KUKA KRL program: MyProgram_279().src

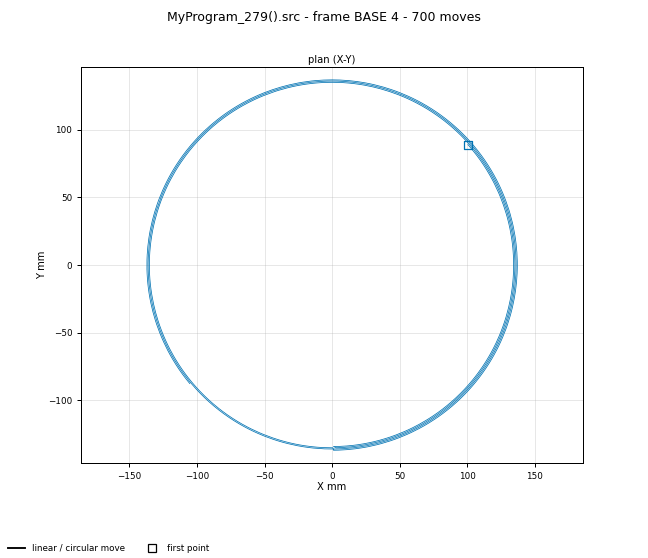
[picture p0: tool path of MyProgram_279().src in frame BASE 4, 700 of 700 moves have a stored position in this frame; points joined in program order, loops and branches not executed]
&ACCESS RVP
&REL 1
&PARAM TEMPLATE = C:\KRC\Roboter\Template\vorgabe
&PARAM EDITMASK = *
DEF MyProgram_279()
; ---- Setting reference (Base) ----
$BASE = BASE_DATA[4]

; --------------------------
; ---- Setting tool (TCP) ----
$TOOL = TOOL_DATA[3]
; --------------------------

$VEL.CP = VEL_APROX_PRINT
Startdeposition()
$VEL.CP = VEL_PRINT
LIN {X 100.485,Y 89.1473,Z 173,A 42.0172,B 8.5894,C 0.1342,E1 8.7113,E2 409.55} C_DIS
LIN {X 102.9839,Y 86.2482,Z 173,A 40.2493,B 8.5893,C 0.1406,E1 8.7146,E2 411.3348} C_DIS
LIN {X 107.2728,Y 80.8516,Z 173,A 37.5079,B 8.5893,C 0.1431,E1 8.7192,E2 414.0536} C_DIS
LIN {X 109.4869,Y 77.827,Z 173,A 35.923,B 8.5892,C 0.1466,E1 8.7218,E2 415.6375} C_DIS
LIN {X 111.988,Y 74.1839,Z 173,A 34.0395,B 8.5891,C 0.151,E1 8.7248,E2 417.5218} C_DIS
LIN {X 114.278,Y 70.6054,Z 173,A 32.2397,B 8.5891,C 0.1552,E1 8.7274,E2 419.3211} C_DIS
LIN {X 116.5443,Y 66.7977,Z 173,A 30.3906,B 8.5889,C 0.159,E1 8.73,E2 421.1663} C_DIS
LIN {X 118.6905,Y 62.9024,Z 173,A 28.6674,B 8.5889,C 0.1602,E1 8.7323,E2 422.8695} C_DIS
LIN {X 120.2957,Y 59.7744,Z 173,A 27.1057,B 8.5889,C 0.1653,E1 8.7343,E2 424.4396} C_DIS
LIN {X 121.8682,Y 56.4983,Z 173,A 25.7054,B 8.5889,C 0.1662,E1 8.7359,E2 425.8228} C_DIS
LIN {X 123.1677,Y 53.6072,Z 173,A 24.298,B 8.5887,C 0.171,E1 8.7375,E2 427.2377} C_DIS
LIN {X 124.4105,Y 50.6572,Z 173,A 23.0997,B 8.5887,C 0.171,E1 8.7388,E2 428.4167} C_DIS
LIN {X 126.8287,Y 44.2546,Z 173,A 20.1497,B 8.5885,C 0.1796,E1 8.7417,E2 431.3725} C_DIS
LIN {X 127.8957,Y 41.0691,Z 173,A 18.3823,B 8.5883,C 0.1906,E1 8.7432,E2 433.1816} C_DIS
LIN {X 128.857,Y 37.9453,Z 173,A 17.2852,B 8.5883,C 0.1882,E1 8.7441,E2 434.2437} C_DIS
LIN {X 129.7659,Y 34.7098,Z 173,A 15.8546,B 8.5883,C 0.1921,E1 8.7451,E2 435.675} C_DIS
LIN {X 130.7274,Y 30.8976,Z 173,A 14.1088,B 8.5881,C 0.1983,E1 8.7463,E2 437.4306} C_DIS
LIN {X 131.5915,Y 26.9758,Z 173,A 12.5684,B 8.5881,C 0.1994,E1 8.7472,E2 438.9513} C_DIS
LIN {X 132.2101,Y 23.7589,Z 173,A 11.1939,B 8.5881,C 0.2029,E1 8.7479,E2 440.3242} C_DIS
LIN {X 132.7584,Y 20.4746,Z 173,A 9.8483,B 8.588,C 0.2054,E1 8.7485,E2 441.6618} C_DIS
LIN {X 133.24,Y 17.0665,Z 173,A 8.3029,B 8.5878,C 0.2112,E1 8.7491,E2 443.2179} C_DIS
LIN {X 133.6974,Y 13.002,Z 173,A 6.6491,B 8.5878,C 0.2143,E1 8.7496,E2 444.8621} C_DIS
LIN {X 133.9613,Y 9.9205,Z 173,A 5.3303,B 8.5877,C 0.2181,E1 8.7498,E2 446.182} C_DIS
LIN {X 134.1788,Y 6.3448,Z 173,A 3.8957,B 8.5876,C 0.2205,E1 8.7501,E2 447.6065} C_DIS
LIN {X 134.3024,Y 2.6623,Z 173,A 2.2339,B 8.5874,C 0.227,E1 8.7501,E2 449.2808} C_DIS
LIN {X 134.324,Y -1.2062,Z 173,A 0.5555,B 8.5873,C 0.2324,E1 8.7501,E2 450.9642} C_DIS
LIN {X 134.2251,Y -5.2587,Z 173,A -1.0909,B 8.5872,C 0.2356,E1 8.7501,E2 452.602} C_DIS
LIN {X 133.985,Y -9.596,Z 173,A -2.8654,B 8.5871,C 0.2393,E1 8.7497,E2 454.3687} C_DIS
LIN {X 133.6414,Y -13.585,Z 173,A -4.6499,B 8.5869,C 0.2459,E1 8.7493,E2 456.1642} C_DIS
LIN {X 133.1911,Y -17.4395,Z 173,A -6.1529,B 8.5869,C 0.2474,E1 8.7488,E2 457.6502} C_DIS
LIN {X 132.6837,Y -20.9568,Z 173,A -7.6551,B 8.5867,C 0.2515,E1 8.7481,E2 459.1521} C_DIS
LIN {X 131.966,Y -25.0793,Z 173,A -9.4147,B 8.5867,C 0.2561,E1 8.7473,E2 460.9104} C_DIS
LIN {X 131.3008,Y -28.3563,Z 173,A -10.761,B 8.5865,C 0.2584,E1 8.7465,E2 462.2482} C_DIS
LIN {X 130.5715,Y -31.5445,Z 173,A -12.2103,B 8.5864,C 0.2636,E1 8.7456,E2 463.7057} C_DIS
LIN {X 128.6891,Y -38.5187,Z 173,A -15.3512,B 8.5861,C 0.2735,E1 8.7432,E2 466.8571} C_DIS
LIN {X 127.5485,Y -42.1357,Z 173,A -16.8717,B 8.5861,C 0.276,E1 8.7419,E2 468.3673} C_DIS
LIN {X 126.1394,Y -46.1868,Z 173,A -18.7317,B 8.5858,C 0.2817,E1 8.7402,E2 470.2329} C_DIS
LIN {X 124.7098,Y -49.9148,Z 173,A -20.2936,B 8.5858,C 0.2833,E1 8.7386,E2 471.7791} C_DIS
LIN {X 123.4262,Y -53.0093,Z 173,A -21.6078,B 8.5858,C 0.2847,E1 8.7372,E2 473.0806} C_DIS
LIN {X 121.271,Y -57.7684,Z 173,A -24.375,B 8.5851,C 0.3021,E1 8.7338,E2 475.9163} C_DIS
LIN {X 119.2793,Y -61.7811,Z 173,A -25.7267,B 8.5854,C 0.2953,E1 8.7322,E2 477.2014} C_DIS
LIN {X 117.6517,Y -64.8271,Z 173,A -27.5786,B 8.585,C 0.3071,E1 8.7297,E2 479.1015} C_DIS
LIN {X 115.8509,Y -67.9927,Z 173,A -28.7916,B 8.585,C 0.3039,E1 8.728,E2 480.2742} C_DIS
LIN {X 113.7196,Y -71.5006,Z 173,A -30.5786,B 8.5849,C 0.3091,E1 8.7254,E2 482.0674} C_DIS
LIN {X 111.2545,Y -75.2785,Z 173,A -33.0154,B 8.5843,C 0.3245,E1 8.7215,E2 484.5691} C_DIS
LIN {X 108.269,Y -79.5126,Z 173,A -34.9644,B 8.5843,C 0.3245,E1 8.7183,E2 486.4884} C_DIS
LIN {X 105.8625,Y -82.6903,Z 173,A -36.3361,B 8.5844,C 0.3216,E1 8.716,E2 487.8214} C_DIS
LIN {X 103.7415,Y -85.3365,Z 173,A -37.6368,B 8.5844,C 0.3219,E1 8.7138,E2 489.1056} C_DIS
LIN {X 100.7739,Y -88.8205,Z 173,A -39.6561,B 8.5842,C 0.3277,E1 8.7101,E2 491.1352} C_DIS
LIN {X 97.9294,Y -91.9476,Z 173,A -41.4693,B 8.584,C 0.3319,E1 8.7066,E2 492.9514} C_DIS
LIN {X 94.9858,Y -94.9858,Z 173,A -43.1042,B 8.584,C 0.3322,E1 8.7035,E2 494.5671} C_DIS
LIN {X 91.8309,Y -98.0391,Z 173,A -45.1099,B 8.5838,C 0.3389,E1 8.6994,E2 496.5911} C_DIS
LIN {X 88.4514,Y -101.098,Z 173,A -47.0097,B 8.5837,C 0.3418,E1 8.6954,E2 498.4872} C_DIS
LIN {X 84.9527,Y -104.0551,Z 173,A -48.6273,B 8.5837,C 0.3387,E1 8.6921,E2 500.065} C_DIS
LIN {X 81.7579,Y -106.5834,Z 173,A -50.7305,B 8.5833,C 0.3495,E1 8.6873,E2 502.2152} C_DIS
LIN {X 78.4256,Y -109.0596,Z 173,A -52.5118,B 8.5833,C 0.3529,E1 8.6833,E2 503.9994} C_DIS
LIN {X 74.2386,Y -111.9519,Z 173,A -54.5479,B 8.5832,C 0.3539,E1 8.6786,E2 506.0209} C_DIS
LIN {X 70.5082,Y -114.3377,Z 173,A -56.5951,B 8.5829,C 0.3601,E1 8.6737,E2 508.0893} C_DIS
LIN {X 64.3845,Y -117.8942,Z 173,A -59.5316,B 8.5828,C 0.3631,E1 8.6666,E2 511.018} C_DIS
LIN {X 59.9186,Y -120.2246,Z 173,A -61.4357,B 8.5828,C 0.3613,E1 8.6619,E2 512.8936} C_DIS
LIN {X 56.6377,Y -121.8037,Z 173,A -62.9476,B 8.5828,C 0.3625,E1 8.6581,E2 514.4015} C_DIS
LIN {X 53.5188,Y -123.2059,Z 173,A -64.428,B 8.5828,C 0.3648,E1 8.6543,E2 515.8858} C_DIS
LIN {X 50.3544,Y -124.5326,Z 173,A -65.8538,B 8.5827,C 0.3658,E1 8.6507,E2 517.3081} C_DIS
LIN {X 47.4368,Y -125.6733,Z 173,A -67.113,B 8.5827,C 0.3658,E1 8.6474,E2 518.5588} C_DIS
LIN {X 43.2176,Y -127.1882,Z 173,A -69.2595,B 8.5824,C 0.3725,E1 8.6417,E2 520.736} C_DIS
LIN {X 39.3019,Y -128.4496,Z 173,A -70.9006,B 8.5824,C 0.372,E1 8.6373,E2 522.3641} C_DIS
LIN {X 35.3098,Y -129.6059,Z 173,A -72.676,B 8.5824,C 0.3737,E1 8.6326,E2 524.1412} C_DIS
LIN {X 31.6272,Y -130.5515,Z 173,A -74.2847,B 8.5823,C 0.3748,E1 8.6282,E2 525.7494} C_DIS
LIN {X 27.725,Y -131.437,Z 173,A -75.9912,B 8.5823,C 0.376,E1 8.6235,E2 527.4569} C_DIS
LIN {X 23.8324,Y -132.1969,Z 173,A -77.6907,B 8.5822,C 0.3773,E1 8.6189,E2 529.1585} C_DIS
LIN {X 19.6935,Y -132.8783,Z 173,A -79.4646,B 8.5822,C 0.378,E1 8.614,E2 530.9316} C_DIS
LIN {X 15.995,Y -133.3723,Z 173,A -81.0275,B 8.5822,C 0.3782,E1 8.6097,E2 532.4918} C_DIS
LIN {X 10.8636,Y -133.8887,Z 173,A -83.2675,B 8.5821,C 0.3799,E1 8.6034,E2 534.7381} C_DIS
LIN {X 4.7872,Y -134.2435,Z 173,A -85.8421,B 8.5821,C 0.3802,E1 8.5962,E2 537.3113} C_DIS
LIN {X 0.9731,Y -134.3248,Z 173,A -87.1721,B 8.5823,C 0.3749,E1 8.5926,E2 538.6052} C_DIS
Enddeposition()
LIN {X 0.9731,Y -134.3248,Z 173,A -87.1721,B 8.5823,C 0.3749,E1 8.5926,E2 538.6052} C_DIS
Startdeposition()
$VEL.CP = VEL_PRINT
LIN {X 3.1797,Y -135.2005,Z 173,A -85.0351,B 8.4211,C 0.3601,E1 8.4372,E2 536.3964} C_DIS
LIN {X 8.6007,Y -134.9631,Z 173,A -83.5881,B 8.4204,C 0.3756,E1 8.4409,E2 535.0567} C_DIS
LIN {X 14.6467,Y -134.4411,Z 173,A -80.9054,B 8.4206,C 0.3725,E1 8.4484,E2 532.3585} C_DIS
LIN {X 18.2658,Y -133.9991,Z 173,A -79.1927,B 8.4208,C 0.3685,E1 8.4532,E2 530.6237} C_DIS
LIN {X 22.5658,Y -133.3408,Z 173,A -77.3912,B 8.4208,C 0.3682,E1 8.4581,E2 528.8263} C_DIS
LIN {X 26.9688,Y -132.52,Z 173,A -75.6345,B 8.4208,C 0.3697,E1 8.4629,E2 527.0862} C_DIS
LIN {X 30.1469,Y -131.8334,Z 173,A -74.2295,B 8.4208,C 0.3681,E1 8.4667,E2 525.6768} C_DIS
LIN {X 33.3306,Y -131.0646,Z 173,A -72.832,B 8.4208,C 0.3668,E1 8.4705,E2 524.2772} C_DIS
LIN {X 37.4094,Y -129.9606,Z 173,A -71.0032,B 8.4209,C 0.3644,E1 8.4755,E2 522.4423} C_DIS
LIN {X 41.0365,Y -128.8598,Z 173,A -69.4333,B 8.4209,C 0.3636,E1 8.4796,E2 520.8757} C_DIS
LIN {X 45.0729,Y -127.5065,Z 173,A -67.7068,B 8.4209,C 0.3632,E1 8.4842,E2 519.1578} C_DIS
LIN {X 48.3644,Y -126.294,Z 173,A -66.2819,B 8.421,C 0.3627,E1 8.4879,E2 517.7394} C_DIS
LIN {X 50.929,Y -125.2805,Z 173,A -65.0721,B 8.421,C 0.3605,E1 8.491,E2 516.5235} C_DIS
LIN {X 53.8536,Y -124.0509,Z 173,A -63.7005,B 8.4212,C 0.3583,E1 8.4946,E2 515.1473} C_DIS
LIN {X 57.7786,Y -122.2733,Z 173,A -62.0162,B 8.4212,C 0.3587,E1 8.4988,E2 513.4794} C_DIS
LIN {X 61.6591,Y -120.3622,Z 173,A -60.1136,B 8.4213,C 0.3547,E1 8.5036,E2 511.5664} C_DIS
LIN {X 66.6135,Y -117.6943,Z 173,A -57.6159,B 8.4216,C 0.3489,E1 8.5097,E2 509.0523} C_DIS
LIN {X 70.7017,Y -115.2849,Z 173,A -55.6539,B 8.4216,C 0.3467,E1 8.5144,E2 507.0947} C_DIS
LIN {X 74.6014,Y -112.8009,Z 173,A -53.7083,B 8.4218,C 0.3437,E1 8.519,E2 505.1492} C_DIS
LIN {X 78.6189,Y -110.0383,Z 173,A -51.7429,B 8.4218,C 0.3421,E1 8.5235,E2 503.1945} C_DIS
LIN {X 81.7657,Y -107.7212,Z 173,A -49.6484,B 8.4223,C 0.3301,E1 8.5283,E2 501.0428} C_DIS
LIN {X 85.0887,Y -105.1157,Z 173,A -48.2843,B 8.4221,C 0.3354,E1 8.5311,E2 499.731} C_DIS
LIN {X 88.4159,Y -102.3328,Z 173,A -46.4652,B 8.4223,C 0.3322,E1 8.535,E2 497.9126} C_DIS
LIN {X 91.7629,Y -99.3429,Z 173,A -44.5493,B 8.4224,C 0.3281,E1 8.5389,E2 495.993} C_DIS
LIN {X 95.6283,Y -95.6283,Z 173,A -42.418,B 8.4224,C 0.3262,E1 8.5432,E2 493.8773} C_DIS
LIN {X 98.3275,Y -92.8496,Z 173,A -40.7262,B 8.4227,C 0.3216,E1 8.5465,E2 492.1774} C_DIS
LIN {X 101.0457,Y -89.8848,Z 173,A -39.0307,B 8.4227,C 0.318,E1 8.5496,E2 490.4813} C_DIS
LIN {X 104.5568,Y -85.7745,Z 173,A -36.7353,B 8.423,C 0.3127,E1 8.5538,E2 488.183} C_DIS
LIN {X 108.0978,Y -81.2666,Z 173,A -34.3605,B 8.4232,C 0.3081,E1 8.5578,E2 485.8126} C_DIS
LIN {X 111.5883,Y -76.403,Z 173,A -32.212,B 8.4231,C 0.3101,E1 8.5612,E2 483.7105} C_DIS
LIN {X 114.2276,Y -72.398,Z 173,A -29.8489,B 8.4235,C 0.2981,E1 8.5649,E2 481.3037} C_DIS
LIN {X 116.5329,Y -68.6255,Z 173,A -27.7284,B 8.4239,C 0.2881,E1 8.5679,E2 479.1499} C_DIS
LIN {X 118.4042,Y -65.344,Z 173,A -26.6704,B 8.4236,C 0.2955,E1 8.5693,E2 478.1588} C_DIS
LIN {X 119.9038,Y -62.5461,Z 173,A -25.1858,B 8.4238,C 0.289,E1 8.5713,E2 476.6552} C_DIS
LIN {X 121.4823,Y -59.4226,Z 173,A -22.9203,B 8.4245,C 0.2684,E1 8.5742,E2 474.2889} C_DIS
LIN {X 124.0675,Y -53.8154,Z 173,A -21.4335,B 8.424,C 0.2855,E1 8.5757,E2 472.9424} C_DIS
LIN {X 125.5947,Y -50.1496,Z 173,A -19.5623,B 8.4242,C 0.277,E1 8.5777,E2 471.0459} C_DIS
LIN {X 126.6911,Y -47.3097,Z 173,A -18.1837,B 8.4244,C 0.2715,E1 8.5791,E2 469.6547} C_DIS
LIN {X 127.9892,Y -43.681,Z 173,A -16.684,B 8.4244,C 0.2699,E1 8.5804,E2 468.1702} C_DIS
LIN {X 128.9127,Y -40.871,Z 173,A -15.3598,B 8.4246,C 0.2648,E1 8.5816,E2 466.8357} C_DIS
LIN {X 130.0092,Y -37.2433,Z 173,A -13.0796,B 8.4252,C 0.2458,E1 8.5834,E2 464.4687} C_DIS
LIN {X 131.459,Y -31.7395,Z 173,A -11.7613,B 8.4247,C 0.2625,E1 8.5842,E2 463.2858} C_DIS
LIN {X 132.4574,Y -27.2767,Z 173,A -9.5172,B 8.4251,C 0.2504,E1 8.5856,E2 461.0015} C_DIS
LIN {X 133.2044,Y -23.3604,Z 173,A -7.7659,B 8.4252,C 0.2443,E1 8.5864,E2 459.2407} C_DIS
LIN {X 133.8801,Y -19.1054,Z 173,A -6.0865,B 8.4253,C 0.2422,E1 8.5871,E2 457.5779} C_DIS
LIN {X 134.3319,Y -15.6208,Z 173,A -4.6379,B 8.4253,C 0.2387,E1 8.5876,E2 456.1329} C_DIS
LIN {X 134.7345,Y -11.6447,Z 173,A -2.9675,B 8.4255,C 0.2343,E1 8.5881,E2 454.4637} C_DIS
LIN {X 134.9923,Y -8.1275,Z 173,A -1.3919,B 8.4257,C 0.2282,E1 8.5884,E2 452.8765} C_DIS
LIN {X 135.1862,Y -3.6953,Z 173,A 0.338,B 8.4257,C 0.226,E1 8.5885,E2 451.1636} C_DIS
LIN {X 135.2394,Y 0.1311,Z 173,A 2.0503,B 8.4259,C 0.2194,E1 8.5885,E2 449.4386} C_DIS
LIN {X 135.1662,Y 4.4152,Z 173,A 3.7592,B 8.4259,C 0.2164,E1 8.5885,E2 447.7414} C_DIS
LIN {X 134.9832,Y 8.2747,Z 173,A 5.3221,B 8.4261,C 0.2132,E1 8.5882,E2 446.1862} C_DIS
LIN {X 134.7234,Y 11.7761,Z 173,A 6.8793,B 8.4262,C 0.2075,E1 8.5878,E2 444.619} C_DIS
LIN {X 134.2911,Y 15.9626,Z 173,A 8.5658,B 8.4262,C 0.2044,E1 8.5873,E2 442.943} C_DIS
LIN {X 133.7903,Y 19.734,Z 173,A 10.2222,B 8.4264,C 0.1989,E1 8.5867,E2 441.2797} C_DIS
LIN {X 133.1155,Y 23.8569,Z 173,A 11.8788,B 8.4264,C 0.1962,E1 8.5859,E2 439.6358} C_DIS
LIN {X 132.477,Y 27.1805,Z 173,A 13.2505,B 8.4266,C 0.1935,E1 8.5852,E2 438.2706} C_DIS
LIN {X 131.6646,Y 30.8858,Z 173,A 14.9649,B 8.4267,C 0.1867,E1 8.5841,E2 436.5417} C_DIS
LIN {X 130.706,Y 34.7103,Z 173,A 16.4987,B 8.4267,C 0.1849,E1 8.583,E2 435.0236} C_DIS
LIN {X 129.7458,Y 38.1432,Z 173,A 18.322,B 8.427,C 0.1741,E1 8.5816,E2 433.1602} C_DIS
LIN {X 128.6869,Y 41.578,Z 173,A 19.5895,B 8.427,C 0.1754,E1 8.5805,E2 431.9235} C_DIS
LIN {X 126.9178,Y 46.6997,Z 173,A 22.0901,B 8.4272,C 0.1648,E1 8.5781,E2 429.3957} C_DIS
LIN {X 125.6176,Y 50.0929,Z 173,A 23.1235,B 8.427,C 0.1714,E1 8.5772,E2 428.4242} C_DIS
LIN {X 123.9922,Y 53.9895,Z 173,A 24.9665,B 8.4271,C 0.1655,E1 8.5751,E2 426.5732} C_DIS
LIN {X 122.6804,Y 56.9065,Z 173,A 26.3336,B 8.4272,C 0.1617,E1 8.5735,E2 425.2039} C_DIS
LIN {X 121.1858,Y 60.0236,Z 173,A 27.7918,B 8.4272,C 0.158,E1 8.5718,E2 423.7455} C_DIS
LIN {X 119.6303,Y 63.0669,Z 173,A 29.1984,B 8.4273,C 0.1552,E1 8.57,E2 422.3432} C_DIS
LIN {X 117.6594,Y 66.6765,Z 173,A 31.0566,B 8.4275,C 0.1484,E1 8.5674,E2 420.4698} C_DIS
LIN {X 115.435,Y 70.457,Z 173,A 32.8581,B 8.4275,C 0.1451,E1 8.5648,E2 418.6744} C_DIS
LIN {X 113.1585,Y 74.0582,Z 173,A 34.6628,B 8.4275,C 0.1407,E1 8.5621,E2 416.8687} C_DIS
LIN {X 110.5824,Y 77.8516,Z 173,A 36.3712,B 8.4275,C 0.141,E1 8.5594,E2 415.1882} C_DIS
LIN {X 108.5001,Y 80.7283,Z 173,A 38.0366,B 8.4277,C 0.1342,E1 8.5566,E2 413.5023} C_DIS
LIN {X 104.2889,Y 86.1,Z 173,A 40.7446,B 8.4277,C 0.1315,E1 8.552,E2 410.8158} C_DIS
LIN {X 101.8703,Y 88.9481,Z 173,A 42.4537,B 8.4278,C 0.1255,E1 8.5488,E2 409.0907} C_DIS
LIN {X 98.7737,Y 92.3752,Z 173,A 44.3706,B 8.4278,C 0.1221,E1 8.5452,E2 407.178} C_DIS
LIN {X 95.502,Y 95.7537,Z 173,A 46.2585,B 8.4279,C 0.1202,E1 8.5415,E2 405.3023} C_DIS
LIN {X 92.5535,Y 98.6068,Z 173,A 48.0619,B 8.4279,C 0.1154,E1 8.5379,E2 403.4904} C_DIS
LIN {X 89.182,Y 101.6663,Z 173,A 49.991,B 8.428,C 0.1118,E1 8.5339,E2 401.5607} C_DIS
LIN {X 85.7804,Y 104.552,Z 173,A 51.8548,B 8.428,C 0.1088,E1 8.5299,E2 399.6997} C_DIS
LIN {X 82.3114,Y 107.3043,Z 173,A 53.6976,B 8.428,C 0.1062,E1 8.5258,E2 397.8607} C_DIS
LIN {X 78.8304,Y 109.887,Z 173,A 55.5035,B 8.4281,C 0.1037,E1 8.5217,E2 396.0582} C_DIS
LIN {X 74.0069,Y 113.1923,Z 173,A 57.9951,B 8.4281,C 0.0995,E1 8.516,E2 393.5646} C_DIS
LIN {X 70.2078,Y 115.5867,Z 173,A 59.8837,B 8.4282,C 0.0969,E1 8.5115,E2 391.6775} C_DIS
LIN {X 66.4641,Y 117.7791,Z 173,A 61.6957,B 8.4282,C 0.0948,E1 8.5071,E2 389.8686} C_DIS
LIN {X 62.5875,Y 119.882,Z 173,A 63.4373,B 8.4282,C 0.0948,E1 8.5029,E2 388.1424} C_DIS
LIN {X 59.215,Y 121.5847,Z 173,A 65.0144,B 8.4282,C 0.0931,E1 8.4989,E2 386.5682} C_DIS
LIN {X 55.8747,Y 123.1557,Z 173,A 66.6829,B 8.4282,C 0.0893,E1 8.4946,E2 384.887} C_DIS
LIN {X 52.258,Y 124.7314,Z 173,A 68.2626,B 8.4282,C 0.0891,E1 8.4906,E2 383.3186} C_DIS
LIN {X 49.0309,Y 126.0349,Z 173,A 69.5241,B 8.4282,C 0.0916,E1 8.4874,E2 382.0831} C_DIS
LIN {X 45.1831,Y 127.467,Z 173,A 71.4243,B 8.4283,C 0.0869,E1 8.4824,E2 380.1637} C_DIS
LIN {X 42.4832,Y 128.3903,Z 173,A 72.6443,B 8.4283,C 0.0856,E1 8.4791,E2 378.9424} C_DIS
LIN {X 35.937,Y 130.375,Z 173,A 75.4831,B 8.4283,C 0.0844,E1 8.4716,E2 376.1115} C_DIS
LIN {X 33.1168,Y 131.1189,Z 173,A 76.7176,B 8.4283,C 0.0835,E1 8.4682,E2 374.8774} C_DIS
LIN {X 30.0725,Y 131.8504,Z 173,A 78.0472,B 8.4283,C 0.0826,E1 8.4646,E2 373.5477} C_DIS
LIN {X 26.8953,Y 132.535,Z 173,A 79.4292,B 8.4283,C 0.0817,E1 8.4608,E2 372.1655} C_DIS
LIN {X 23.7507,Y 133.1345,Z 173,A 80.8155,B 8.4283,C 0.0805,E1 8.457,E2 370.7759} C_DIS
LIN {X 20.398,Y 133.6896,Z 173,A 82.2229,B 8.4283,C 0.0805,E1 8.4531,E2 369.3729} C_DIS
LIN {X 16.3594,Y 134.2438,Z 173,A 84.0058,B 8.4283,C 0.0788,E1 8.4482,E2 367.5838} C_DIS
LIN {X 12.3179,Y 134.6758,Z 173,A 85.7905,B 8.4284,C 0.0772,E1 8.4432,E2 365.7921} C_DIS
LIN {X 8.2747,Y 134.9832,Z 173,A 87.3954,B 8.4284,C 0.0789,E1 8.4388,E2 364.2016} C_DIS
LIN {X 4.6219,Y 135.1592,Z 173,A 89.0917,B 8.4284,C 0.0762,E1 8.434,E2 362.4881} C_DIS
LIN {X 0.4143,Y 135.2365,Z 173,A 90.7128,B 8.4284,C 0.079,E1 8.4295,E2 360.8875} C_DIS
LIN {X -3.2674,Y 135.1981,Z 173,A 92.3499,B 8.4284,C 0.0778,E1 8.4249,E2 359.2418} C_DIS
LIN {X -7.2879,Y 135.041,Z 173,A 94.0757,B 8.4284,C 0.0776,E1 8.4201,E2 357.5143} C_DIS
LIN {X -11.2924,Y 134.7643,Z 173,A 95.6702,B 8.4284,C 0.0799,E1 8.4157,E2 355.9335} C_DIS
LIN {X -14.7888,Y 134.4259,Z 173,A 97.2629,B 8.4284,C 0.0785,E1 8.4113,E2 354.3289} C_DIS
LIN {X -18.986,Y 133.8972,Z 173,A 98.9835,B 8.4284,C 0.0805,E1 8.4065,E2 352.618} C_DIS
LIN {X -22.2797,Y 133.3886,Z 173,A 100.3841,B 8.4284,C 0.0814,E1 8.4027,E2 351.2196} C_DIS
LIN {X -25.5723,Y 132.7967,Z 173,A 101.8299,B 8.4284,C 0.0816,E1 8.3987,E2 349.7713} C_DIS
LIN {X -29.4458,Y 131.9935,Z 173,A 103.6301,B 8.4284,C 0.0806,E1 8.3937,E2 347.9571} C_DIS
LIN {X -33.2572,Y 131.0832,Z 173,A 105.1705,B 8.4284,C 0.0838,E1 8.3896,E2 346.4322} C_DIS
LIN {X -39.8741,Y 129.2246,Z 173,A 107.7166,B 8.4283,C 0.0923,E1 8.3829,E2 343.9324} C_DIS
LIN {X -42.3962,Y 128.4193,Z 173,A 109.2843,B 8.4283,C 0.0859,E1 8.3786,E2 342.3117} C_DIS
LIN {X -50.6496,Y 125.3932,Z 173,A 112.9805,B 8.4283,C 0.0902,E1 8.3689,E2 338.6218} C_DIS
LIN {X -54.0091,Y 123.9837,Z 173,A 114.5342,B 8.4283,C 0.0918,E1 8.3649,E2 337.0681} C_DIS
LIN {X -57.547,Y 122.384,Z 173,A 116.7812,B 8.4283,C 0.0839,E1 8.3591,E2 334.7493} C_DIS
LIN {X -61.773,Y 120.3037,Z 173,A 118.3745,B 8.4283,C 0.0932,E1 8.3552,E2 333.2066} C_DIS
LIN {X -66.2426,Y 117.9036,Z 173,A 120.752,B 8.4283,C 0.0925,E1 8.3494,E2 330.8032} C_DIS
LIN {X -69.4915,Y 116.0187,Z 173,A 122.0217,B 8.4282,C 0.1001,E1 8.3464,E2 329.5739} C_DIS
LIN {X -73.0138,Y 113.8347,Z 173,A 123.7999,B 8.4282,C 0.1025,E1 8.3422,E2 327.7946} C_DIS
LIN {X -76.4463,Y 111.5585,Z 173,A 125.9689,B 8.4282,C 0.0985,E1 8.3371,E2 325.5756} C_DIS
LIN {X -79.7958,Y 109.1873,Z 173,A 127.4535,B 8.4281,C 0.1056,E1 8.3338,E2 324.1234} C_DIS
LIN {X -84.2142,Y 105.8173,Z 173,A 129.7481,B 8.4281,C 0.1108,E1 8.3288,E2 321.8383} C_DIS
LIN {X -87.7892,Y 102.8711,Z 173,A 132.0045,B 8.4281,C 0.1098,E1 8.3239,E2 319.548} C_DIS
LIN {X -90.5457,Y 100.4533,Z 173,A 133.1644,B 8.4279,C 0.1191,E1 8.3216,E2 318.4374} C_DIS
LIN {X -93.2303,Y 97.9667,Z 173,A 134.8712,B 8.4279,C 0.1197,E1 8.3181,E2 316.7131} C_DIS
LIN {X -96.2981,Y 94.9534,Z 173,A 136.7066,B 8.4279,C 0.1233,E1 8.3144,E2 314.8778} C_DIS
LIN {X -99.6578,Y 91.4204,Z 173,A 138.841,B 8.4279,C 0.1266,E1 8.3103,E2 312.737} C_DIS
LIN {X -102.769,Y 87.9086,Z 173,A 140.7675,B 8.4277,C 0.1319,E1 8.3068,E2 310.8199} C_DIS
LIN {X -105.5058,Y 84.6051,Z 173,A 142.6514,B 8.4277,C 0.135,E1 8.3035,E2 308.9297} C_DIS
LIN {X -108.2156,Y 81.1104,Z 173,A 144.5995,B 8.4277,C 0.1382,E1 8.3002,E2 306.9744} C_DIS
LIN {X -111.7506,Y 76.1664,Z 173,A 147.0901,B 8.4275,C 0.1457,E1 8.2962,E2 304.4967} C_DIS
LIN {X -114.0158,Y 72.731,Z 173,A 148.9801,B 8.4275,C 0.1477,E1 8.2933,E2 302.5906} C_DIS
LIN {X -116.0676,Y 69.4096,Z 173,A 150.4747,B 8.4274,C 0.1542,E1 8.2912,E2 301.1171} C_DIS
LIN {X -119.5933,Y 63.1373,Z 173,A 153.4127,B 8.4272,C 0.1637,E1 8.2872,E2 298.1957} C_DIS
LIN {X -121.399,Y 59.5915,Z 173,A 155.3779,B 8.4272,C 0.1638,E1 8.2847,E2 296.1982} C_DIS
LIN {X -122.7688,Y 56.7152,Z 173,A 156.7708,B 8.4272,C 0.1668,E1 8.2831,E2 294.8014} C_DIS
LIN {X -124.2485,Y 53.3966,Z 173,A 158.268,B 8.427,C 0.1715,E1 8.2814,E2 293.3109} C_DIS
LIN {X -125.7375,Y 49.7953,Z 173,A 160.2796,B 8.427,C 0.1705,E1 8.2792,E2 291.257} C_DIS
LIN {X -126.9135,Y 46.7131,Z 173,A 161.8612,B 8.427,C 0.1716,E1 8.2777,E2 289.6541} C_DIS
LIN {X -128.29,Y 42.7846,Z 173,A 163.1946,B 8.4268,C 0.1829,E1 8.2766,E2 288.3752} C_DIS
LIN {X -129.3538,Y 39.4519,Z 173,A 164.6848,B 8.4267,C 0.1869,E1 8.2753,E2 286.8856} C_DIS
LIN {X -130.4603,Y 35.6314,Z 173,A 166.3686,B 8.4266,C 0.1916,E1 8.2741,E2 285.2036} C_DIS
LIN {X -131.2034,Y 32.7838,Z 173,A 167.5985,B 8.4266,C 0.1954,E1 8.2732,E2 283.977} C_DIS
LIN {X -131.8991,Y 29.859,Z 173,A 168.9379,B 8.4264,C 0.198,E1 8.2724,E2 282.6307} C_DIS
LIN {X -132.7237,Y 25.9542,Z 173,A 170.7097,B 8.4264,C 0.2016,E1 8.2714,E2 280.8508} C_DIS
LIN {X -133.5224,Y 21.4778,Z 173,A 172.6118,B 8.4262,C 0.2075,E1 8.2705,E2 278.9536} C_DIS
LIN {X -134.1105,Y 17.4157,Z 173,A 174.3929,B 8.4262,C 0.2119,E1 8.2698,E2 277.1689} C_DIS
LIN {X -134.5053,Y 14.0502,Z 173,A 175.9725,B 8.4261,C 0.2139,E1 8.2693,E2 275.573} C_DIS
LIN {X -134.8812,Y 9.7977,Z 173,A 177.71,B 8.4259,C 0.2201,E1 8.2689,E2 273.846} C_DIS
LIN {X -135.1139,Y 5.7843,Z 173,A 179.5245,B 8.4259,C 0.2234,E1 8.2687,E2 272.0194} C_DIS
LIN {X -135.2305,Y 1.4907,Z 173,A -178.6249,B 8.4257,C 0.2282,E1 8.2686,E2 270.1666} C_DIS
LIN {X -135.2093,Y -2.7701,Z 173,A -176.8534,B 8.4255,C 0.2339,E1 8.2686,E2 268.4009} C_DIS
LIN {X -135.0708,Y -6.6957,Z 173,A -175.1199,B 8.4255,C 0.2377,E1 8.2688,E2 266.6603} C_DIS
LIN {X -134.827,Y -10.5403,Z 173,A -173.3942,B 8.4253,C 0.241,E1 8.2692,E2 264.9246} C_DIS
LIN {X -134.4653,Y -14.4223,Z 173,A -171.8086,B 8.4252,C 0.2467,E1 8.2696,E2 263.3484} C_DIS
LIN {X -134.0773,Y -17.669,Z 173,A -170.4011,B 8.4251,C 0.2504,E1 8.2701,E2 261.9394} C_DIS
LIN {X -133.4689,Y -21.7982,Z 173,A -168.5618,B 8.4249,C 0.2543,E1 8.2709,E2 260.0928} C_DIS
LIN {X -132.5791,Y -26.6787,Z 173,A -166.6981,B 8.4247,C 0.2639,E1 8.2719,E2 258.2601} C_DIS
LIN {X -132.1083,Y -28.9208,Z 173,A -165.4686,B 8.4247,C 0.2627,E1 8.2726,E2 256.9995} C_DIS
LIN {X -130.6198,Y -35.0338,Z 173,A -162.6318,B 8.4245,C 0.2675,E1 8.2745,E2 254.1435} C_DIS
LIN {X -128.7655,Y -41.3318,Z 173,A -159.9388,B 8.4243,C 0.2765,E1 8.2767,E2 251.4637} C_DIS
LIN {X -127.5665,Y -44.9001,Z 173,A -158.2412,B 8.4242,C 0.2793,E1 8.2783,E2 249.7545} C_DIS
LIN {X -126.0742,Y -48.9297,Z 173,A -156.4372,B 8.424,C 0.2844,E1 8.28,E2 247.9537} C_DIS
LIN {X -124.6963,Y -52.3421,Z 173,A -154.8858,B 8.4238,C 0.2886,E1 8.2817,E2 246.4043} C_DIS
LIN {X -123.1394,Y -55.9114,Z 173,A -152.8264,B 8.4239,C 0.2866,E1 8.2841,E2 244.2951} C_DIS
LIN {X -121.558,Y -59.2691,Z 173,A -151.7114,B 8.4235,C 0.2977,E1 8.2854,E2 243.238} C_DIS
LIN {X -120.0013,Y -62.3604,Z 173,A -149.3932,B 8.4239,C 0.2882,E1 8.2885,E2 240.8142} C_DIS
LIN {X -117.2998,Y -67.3069,Z 173,A -147.8587,B 8.4232,C 0.3074,E1 8.2905,E2 239.3878} C_DIS
LIN {X -115.6958,Y -70.0273,Z 173,A -146.2667,B 8.4232,C 0.3067,E1 8.2928,E2 237.765} C_DIS
LIN {X -113.3031,Y -73.8363,Z 173,A -143.9413,B 8.4232,C 0.3046,E1 8.2964,E2 235.388} C_DIS
LIN {X -110.9645,Y -77.3061,Z 173,A -142.7004,B 8.4228,C 0.3172,E1 8.2983,E2 234.2146} C_DIS
LIN {X -108.9671,Y -80.097,Z 173,A -140.7825,B 8.423,C 0.3131,E1 8.3015,E2 232.2394} C_DIS
LIN {X -106.7923,Y -82.9745,Z 173,A -139.5121,B 8.4227,C 0.3206,E1 8.3036,E2 231.0019} C_DIS
LIN {X -103.9626,Y -86.494,Z 173,A -137.5595,B 8.4226,C 0.3242,E1 8.3071,E2 229.0452} C_DIS
LIN {X -100.9881,Y -89.9493,Z 173,A -135.7878,B 8.4223,C 0.3308,E1 8.3103,E2 227.2942} C_DIS
LIN {X -98.2244,Y -92.9589,Z 173,A -134.1406,B 8.4221,C 0.3357,E1 8.3134,E2 225.6581} C_DIS
LIN {X -94.6894,Y -96.557,Z 173,A -131.8092,B 8.4221,C 0.3368,E1 8.318,E2 223.3031} C_DIS
LIN {X -91.6014,Y -99.4914,Z 173,A -129.8629,B 8.4221,C 0.3379,E1 8.322,E2 221.3395} C_DIS
LIN {X -88.2878,Y -102.4432,Z 173,A -127.959,B 8.4219,C 0.341,E1 8.326,E2 219.4332} C_DIS
LIN {X -83.8107,Y -106.1378,Z 173,A -125.716,B 8.4216,C 0.3488,E1 8.3308,E2 217.2178} C_DIS
LIN {X -81.2062,Y -108.1434,Z 173,A -123.626,B 8.422,C 0.3395,E1 8.3357,E2 215.0403} C_DIS
LIN {X -77.5317,Y -110.8075,Z 173,A -122.1468,B 8.4215,C 0.35,E1 8.3389,E2 213.6174} C_DIS
LIN {X -73.9706,Y -113.2159,Z 173,A -120.3116,B 8.4215,C 0.3525,E1 8.3432,E2 211.7807} C_DIS
LIN {X -70.3188,Y -115.5195,Z 173,A -118.4161,B 8.4214,C 0.354,E1 8.3477,E2 209.877} C_DIS
LIN {X -66.5862,Y -117.7105,Z 173,A -116.5571,B 8.4213,C 0.356,E1 8.3522,E2 208.0149} C_DIS
LIN {X -62.6017,Y -119.8746,Z 173,A -114.7615,B 8.4211,C 0.3606,E1 8.3566,E2 206.2351} C_DIS
LIN {X -59.639,Y -121.3756,Z 173,A -113.3573,B 8.4211,C 0.3623,E1 8.3601,E2 204.8312} C_DIS
LIN {X -56.5459,Y -122.8471,Z 173,A -111.8911,B 8.421,C 0.3637,E1 8.3638,E2 203.363} C_DIS
LIN {X -53.8154,Y -124.0675,Z 173,A -110.542,B 8.421,C 0.3636,E1 8.3673,E2 202.0035} C_DIS
LIN {X -50.6716,Y -125.3843,Z 173,A -109.0642,B 8.421,C 0.3644,E1 8.3712,E2 200.5213} C_DIS
LIN {X -46.7701,Y -126.8932,Z 173,A -107.3963,B 8.4208,C 0.3679,E1 8.3755,E2 198.8664} C_DIS
LIN {X -43.9826,Y -127.8846,Z 173,A -105.4921,B 8.4212,C 0.3575,E1 8.3807,E2 196.8796} C_DIS
LIN {X -39.277,Y -129.4073,Z 173,A -104.4405,B 8.4204,C 0.3775,E1 8.3832,E2 195.9596} C_DIS
LIN {X -34.9347,Y -130.6462,Z 173,A -102.0683,B 8.4207,C 0.3706,E1 8.3897,E2 193.5293} C_DIS
LIN {X -31.1899,Y -131.5915,Z 173,A -100.4146,B 8.4207,C 0.3713,E1 8.3942,E2 191.8731} C_DIS
LIN {X -27.335,Y -132.4455,Z 173,A -98.7086,B 8.4207,C 0.3715,E1 8.3989,E2 190.1624} C_DIS
LIN {X -23.9022,Y -133.1074,Z 173,A -97.2871,B 8.4206,C 0.3732,E1 8.4028,E2 188.7479} C_DIS
LIN {X -20.548,Y -133.6664,Z 173,A -95.7481,B 8.4206,C 0.3719,E1 8.407,E2 187.196} C_DIS
LIN {X -16.0004,Y -134.2866,Z 173,A -93.8174,B 8.4206,C 0.3726,E1 8.4124,E2 185.2665} C_DIS
LIN {X -11.1093,Y -134.7798,Z 173,A -91.7973,B 8.4206,C 0.3741,E1 8.418,E2 183.2535} C_DIS
LIN {X -6.4142,Y -135.0849,Z 173,A -89.751,B 8.4206,C 0.3732,E1 8.4237,E2 181.1997} C_DIS
LIN {X 0.5391,Y -135.2358,Z 173,A -87.0998,B 8.4203,C 0.3785,E1 8.431,E2 178.5845} C_DIS
LIN {X 0.5391,Y -135.2358,Z 173,A -87.0998,B 8.4203,C 0.3785,E1 8.431,E2 178.5845} C_DIS
Enddeposition()
LIN {X 0.9633,Y -136.1409,Z 173,A -88.1506,B 8.3746,C 0.4067,E1 8.3832,E2 179.8364} C_DIS
Startdeposition()
$VEL.CP = VEL_PRINT
LIN {X -5.473,Y -136.0352,Z 173,A -89.6005,B 8.3756,C 0.3838,E1 8.3795,E2 181.1295} C_DIS
LIN {X -11.3696,Y -135.6695,Z 173,A -92.4786,B 8.3753,C 0.3908,E1 8.3714,E2 184.0584} C_DIS
LIN {X -14.0067,Y -135.4237,Z 173,A -94.048,B 8.3749,C 0.3988,E1 8.3668,E2 185.6855} C_DIS
LIN {X -18.1324,Y -134.9329,Z 173,A -95.3744,B 8.3753,C 0.3908,E1 8.3633,E2 186.9595} C_DIS
LIN {X -21.6252,Y -134.4189,Z 173,A -97.0144,B 8.3753,C 0.3931,E1 8.3587,E2 188.6194} C_DIS
LIN {X -25.8743,Y -133.664,Z 173,A -98.6972,B 8.3753,C 0.39,E1 8.3541,E2 190.2859} C_DIS
LIN {X -30.1678,Y -132.7605,Z 173,A -100.458,B 8.3755,C 0.3875,E1 8.3494,E2 192.0364} C_DIS
LIN {X -32.929,Y -132.1039,Z 173,A -101.7761,B 8.3755,C 0.3891,E1 8.3457,E2 193.3704} C_DIS
LIN {X -36.51,Y -131.1581,Z 173,A -103.324,B 8.3755,C 0.3879,E1 8.3416,E2 194.9173} C_DIS
LIN {X -40.668,Y -129.9313,Z 173,A -105.4275,B 8.3753,C 0.3914,E1 8.3359,E2 197.0562} C_DIS
LIN {X -43.9343,Y -128.863,Z 173,A -106.619,B 8.3756,C 0.3858,E1 8.3328,E2 198.216} C_DIS
LIN {X -47.2306,Y -127.6909,Z 173,A -108.0585,B 8.3756,C 0.3839,E1 8.329,E2 199.6515} C_DIS
LIN {X -50.0917,Y -126.5972,Z 173,A -109.4673,B 8.3756,C 0.3848,E1 8.3253,E2 201.0756} C_DIS
LIN {X -54.8293,Y -124.6186,Z 173,A -111.6273,B 8.3756,C 0.3826,E1 8.3198,E2 203.2357} C_DIS
LIN {X -58.4419,Y -122.9633,Z 173,A -113.1826,B 8.3759,C 0.3787,E1 8.3159,E2 204.7762} C_DIS
LIN {X -61.5669,Y -121.4286,Z 173,A -114.6935,B 8.3759,C 0.3777,E1 8.3121,E2 206.2929} C_DIS
LIN {X -64.8759,Y -119.6961,Z 173,A -116.3682,B 8.3759,C 0.3775,E1 8.3079,E2 207.9806} C_DIS
LIN {X -68.6334,Y -117.5819,Z 173,A -118.1652,B 8.376,C 0.3748,E1 8.3036,E2 209.7753} C_DIS
LIN {X -72.3367,Y -115.3406,Z 173,A -120.0305,B 8.3761,C 0.3729,E1 8.2991,E2 211.6459} C_DIS
LIN {X -76.0965,Y -112.8951,Z 173,A -121.9348,B 8.3762,C 0.3703,E1 8.2947,E2 213.5521} C_DIS
LIN {X -80.3279,Y -109.9247,Z 173,A -124.1146,B 8.3764,C 0.3669,E1 8.2897,E2 215.7321} C_DIS
LIN {X -83.8425,Y -107.2681,Z 173,A -126.0128,B 8.3764,C 0.3646,E1 8.2855,E2 217.6355} C_DIS
LIN {X -87.8782,Y -103.9879,Z 173,A -128.2297,B 8.3766,C 0.3612,E1 8.2807,E2 219.8554} C_DIS
LIN {X -91.203,Y -101.0844,Z 173,A -130.0393,B 8.3768,C 0.357,E1 8.277,E2 221.6586} C_DIS
LIN {X -94.3736,Y -98.1311,Z 173,A -131.9597,B 8.3769,C 0.3551,E1 8.2731,E2 223.5905} C_DIS
LIN {X -97.6172,Y -94.9045,Z 173,A -133.873,B 8.3771,C 0.351,E1 8.2693,E2 225.5017} C_DIS
LIN {X -100.4642,Y -91.8856,Z 173,A -135.6526,B 8.3771,C 0.348,E1 8.2659,E2 227.2848} C_DIS
LIN {X -103.4597,Y -88.4995,Z 173,A -137.5995,B 8.3773,C 0.3447,E1 8.2623,E2 229.2365} C_DIS
LIN {X -106.1733,Y -85.2246,Z 173,A -139.34,B 8.3775,C 0.34,E1 8.2593,E2 230.9702} C_DIS
LIN {X -108.2797,Y -82.5315,Z 173,A -141.0384,B 8.3775,C 0.3408,E1 8.2563,E2 232.7001} C_DIS
LIN {X -110.2313,Y -79.906,Z 173,A -142.2257,B 8.3777,C 0.3348,E1 8.2544,E2 233.8633} C_DIS
LIN {X -112.4327,Y -76.7782,Z 173,A -144.1202,B 8.3777,C 0.3354,E1 8.2514,E2 235.7923} C_DIS
LIN {X -114.4137,Y -73.7942,Z 173,A -145.4271,B 8.378,C 0.3288,E1 8.2494,E2 237.0736} C_DIS
LIN {X -116.8116,Y -69.9359,Z 173,A -147.3349,B 8.3781,C 0.3241,E1 8.2467,E2 238.9799} C_DIS
LIN {X -118.4981,Y -67.0391,Z 173,A -148.8704,B 8.3782,C 0.3225,E1 8.2445,E2 240.5302} C_DIS
LIN {X -120.606,Y -63.163,Z 173,A -150.6112,B 8.3785,C 0.3161,E1 8.2422,E2 242.2554} C_DIS
LIN {X -122.5946,Y -59.2136,Z 173,A -152.342,B 8.3787,C 0.3094,E1 8.2401,E2 243.969} C_DIS
LIN {X -124.1249,Y -55.9331,Z 173,A -153.9738,B 8.3787,C 0.3071,E1 8.2382,E2 245.6133} C_DIS
LIN {X -125.5351,Y -52.6912,Z 173,A -155.4624,B 8.3789,C 0.3032,E1 8.2366,E2 247.1011} C_DIS
LIN {X -126.6312,Y -50.0043,Z 173,A -156.7674,B 8.3789,C 0.3012,E1 8.2352,E2 248.4156} C_DIS
LIN {X -127.7418,Y -47.0947,Z 173,A -158.0704,B 8.3791,C 0.2976,E1 8.2339,E2 249.7168} C_DIS
LIN {X -129.1425,Y -43.1001,Z 173,A -159.7039,B 8.3794,C 0.2905,E1 8.2324,E2 251.3307} C_DIS
LIN {X -129.8374,Y -40.962,Z 173,A -161.916,B 8.3788,C 0.3068,E1 8.2305,E2 253.6971} C_DIS
LIN {X -131.8402,Y -33.9678,Z 173,A -164.1886,B 8.3795,C 0.2867,E1 8.2289,E2 255.8714} C_DIS
LIN {X -133.0253,Y -28.9788,Z 173,A -166.1746,B 8.3798,C 0.2781,E1 8.2277,E2 257.8346} C_DIS
LIN {X -133.7015,Y -25.6779,Z 173,A -167.6971,B 8.3798,C 0.2756,E1 8.2269,E2 259.3688} C_DIS
LIN {X -134.4917,Y -21.1552,Z 173,A -169.6161,B 8.3801,C 0.2699,E1 8.226,E2 261.2846} C_DIS
LIN {X -135.0007,Y -17.615,Z 173,A -171.0394,B 8.3802,C 0.2644,E1 8.2254,E2 262.6965} C_DIS
LIN {X -135.3176,Y -14.994,Z 173,A -172.2666,B 8.3802,C 0.263,E1 8.2251,E2 263.9372} C_DIS
LIN {X -135.6783,Y -11.2663,Z 173,A -173.8722,B 8.3804,C 0.2589,E1 8.2246,E2 265.545} C_DIS
LIN {X -135.9674,Y -6.9557,Z 173,A -175.7148,B 8.3805,C 0.254,E1 8.2243,E2 267.389} C_DIS
LIN {X -136.1157,Y -2.9061,Z 173,A -177.5396,B 8.3806,C 0.2508,E1 8.2242,E2 269.2269} C_DIS
LIN {X -136.1396,Y 1.4208,Z 173,A -179.3868,B 8.3808,C 0.246,E1 8.2242,E2 271.0757} C_DIS
LIN {X -136.0418,Y 5.3047,Z 173,A 179.0481,B 8.381,C 0.2402,E1 8.2243,E2 272.6306} C_DIS
LIN {X -135.8584,Y 8.8439,Z 173,A 177.39,B 8.381,C 0.2383,E1 8.2246,E2 274.3078} C_DIS
LIN {X -135.5506,Y 12.7123,Z 173,A 176.0005,B 8.3812,C 0.23,E1 8.2249,E2 275.666} C_DIS
LIN {X -135.2226,Y 15.8245,Z 173,A 174.5254,B 8.3812,C 0.2286,E1 8.2254,E2 277.1591} C_DIS
LIN {X -134.7792,Y 19.2362,Z 173,A 173.1239,B 8.3814,C 0.2237,E1 8.2259,E2 278.5536} C_DIS
LIN {X -134.1729,Y 23.0991,Z 173,A 171.2153,B 8.3814,C 0.2229,E1 8.2268,E2 280.4927} C_DIS
LIN {X -133.4586,Y 26.9129,Z 173,A 169.719,B 8.3816,C 0.2162,E1 8.2276,E2 281.9707} C_DIS
LIN {X -132.3811,Y 31.7912,Z 173,A 167.6177,B 8.3818,C 0.2103,E1 8.2289,E2 284.0699} C_DIS
LIN {X -131.6773,Y 34.594,Z 173,A 166.4327,B 8.3818,C 0.2064,E1 8.2297,E2 285.2499} C_DIS
LIN {X -130.8834,Y 37.4909,Z 173,A 164.8651,B 8.3818,C 0.2073,E1 8.2309,E2 286.8533} C_DIS
LIN {X -129.6805,Y 41.453,Z 173,A 163.3835,B 8.382,C 0.1986,E1 8.2321,E2 288.3013} C_DIS
LIN {X -126.6128,Y 50.0517,Z 173,A 159.2289,B 8.3822,C 0.1928,E1 8.2361,E2 292.4903} C_DIS
LIN {X -125.1394,Y 53.6254,Z 173,A 157.8433,B 8.3823,C 0.1848,E1 8.2376,E2 293.8449} C_DIS
LIN {X -123.6632,Y 56.9457,Z 173,A 156.1252,B 8.3823,C 0.1836,E1 8.2396,E2 295.5844} C_DIS
LIN {X -122.2295,Y 59.9615,Z 173,A 154.7265,B 8.3825,C 0.1798,E1 8.2413,E2 296.9809} C_DIS
LIN {X -120.6374,Y 63.1032,Z 173,A 153.0248,B 8.3825,C 0.1793,E1 8.2435,E2 298.7076} C_DIS
LIN {X -118.1392,Y 67.669,Z 173,A 150.8927,B 8.3826,C 0.1728,E1 8.2464,E2 300.8306} C_DIS
LIN {X -115.4877,Y 72.1009,Z 173,A 148.6767,B 8.3826,C 0.1681,E1 8.2496,E2 303.0496} C_DIS
LIN {X -112.9922,Y 75.9529,Z 173,A 146.7043,B 8.3828,C 0.164,E1 8.2526,E2 305.025} C_DIS
LIN {X -110.1789,Y 79.9782,Z 173,A 144.6818,B 8.3828,C 0.1584,E1 8.2559,E2 307.0401} C_DIS
LIN {X -107.5665,Y 83.4587,Z 173,A 142.7977,B 8.3829,C 0.1549,E1 8.2591,E2 308.9286} C_DIS
LIN {X -104.8212,Y 86.8817,Z 173,A 141.0867,B 8.3831,C 0.1487,E1 8.2621,E2 310.6215} C_DIS
LIN {X -102.0063,Y 90.1699,Z 173,A 139.2114,B 8.3831,C 0.1455,E1 8.2655,E2 312.5015} C_DIS
LIN {X -98.6407,Y 93.8403,Z 173,A 136.9253,B 8.3831,C 0.1439,E1 8.2699,E2 314.8087} C_DIS
LIN {X -95.4382,Y 97.0952,Z 173,A 135.3076,B 8.3833,C 0.1353,E1 8.273,E2 316.3878} C_DIS
LIN {X -93.0863,Y 99.3529,Z 173,A 133.6147,B 8.3833,C 0.1375,E1 8.2765,E2 318.1181} C_DIS
LIN {X -90.9115,Y 101.346,Z 173,A 132.1189,B 8.3833,C 0.139,E1 8.2797,E2 319.6434} C_DIS
LIN {X -88.3038,Y 103.6261,Z 173,A 130.8735,B 8.3833,C 0.1329,E1 8.2823,E2 320.862} C_DIS
LIN {X -84.7945,Y 106.5166,Z 173,A 128.9518,B 8.3833,C 0.1296,E1 8.2864,E2 322.7829} C_DIS
LIN {X -81.6088,Y 108.9769,Z 173,A 126.6033,B 8.3833,C 0.1368,E1 8.2919,E2 325.2082} C_DIS
LIN {X -77.1233,Y 112.1958,Z 173,A 124.914,B 8.3835,C 0.123,E1 8.2956,E2 326.8196} C_DIS
LIN {X -73.6702,Y 114.4933,Z 173,A 123.1497,B 8.3835,C 0.1205,E1 8.2997,E2 328.5847} C_DIS
LIN {X -70.0407,Y 116.7491,Z 173,A 121.5279,B 8.3835,C 0.1149,E1 8.3035,E2 330.1836} C_DIS
LIN {X -66.0806,Y 119.0348,Z 173,A 119.3718,B 8.3835,C 0.1159,E1 8.3088,E2 332.3661} C_DIS
LIN {X -62.1513,Y 121.1312,Z 173,A 116.8336,B 8.3835,C 0.124,E1 8.3153,E2 334.9821} C_DIS
LIN {X -57.1445,Y 123.5713,Z 173,A 115.2547,B 8.3837,C 0.1087,E1 8.319,E2 336.4676} C_DIS
LIN {X -54.3368,Y 124.8319,Z 173,A 113.9914,B 8.3837,C 0.1066,E1 8.3222,E2 337.7261} C_DIS
LIN {X -51.762,Y 125.9232,Z 173,A 112.6371,B 8.3837,C 0.1082,E1 8.3258,E2 339.1009} C_DIS
LIN {X -46.6003,Y 127.9218,Z 173,A 110.527,B 8.3837,C 0.1022,E1 8.3312,E2 341.1828} C_DIS
LIN {X -43.4556,Y 129.0241,Z 173,A 108.9069,B 8.3837,C 0.1044,E1 8.3356,E2 342.8282} C_DIS
LIN {X -40.1934,Y 130.077,Z 173,A 107.4346,B 8.3837,C 0.1037,E1 8.3395,E2 344.3031} C_DIS
LIN {X -37.0962,Y 130.9942,Z 173,A 105.9065,B 8.3837,C 0.1054,E1 8.3436,E2 345.8506} C_DIS
LIN {X -32.1239,Y 132.3009,Z 173,A 103.9795,B 8.3837,C 0.0998,E1 8.3488,E2 347.7477} C_DIS
LIN {X -29.3155,Y 132.9526,Z 173,A 102.8523,B 8.3838,C 0.0976,E1 8.3518,E2 348.8637} C_DIS
LIN {X -26.5577,Y 133.5308,Z 173,A 101.4096,B 8.3838,C 0.1013,E1 8.3558,E2 350.3367} C_DIS
LIN {X -22.7999,Y 134.2229,Z 173,A 99.9022,B 8.3838,C 0.0987,E1 8.36,E2 351.8309} C_DIS
LIN {X -19.2283,Y 134.7803,Z 173,A 98.4232,B 8.3838,C 0.0973,E1 8.364,E2 353.304} C_DIS
LIN {X -15.4067,Y 135.2724,Z 173,A 96.8097,B 8.3838,C 0.0966,E1 8.3685,E2 354.9156} C_DIS
LIN {X -11.6178,Y 135.6486,Z 173,A 95.1702,B 8.3838,C 0.0968,E1 8.3731,E2 356.5586} C_DIS
LIN {X -7.4265,Y 135.9437,Z 173,A 93.3296,B 8.3838,C 0.0977,E1 8.3782,E2 358.4071} C_DIS
LIN {X -3.604,Y 136.0976,Z 173,A 91.7853,B 8.3838,C 0.0964,E1 8.3825,E2 359.9427} C_DIS
LIN {X -0.0695,Y 136.1469,Z 173,A 90.1975,B 8.3838,C 0.0981,E1 8.387,E2 361.542} C_DIS
LIN {X 4.1702,Y 136.0819,Z 173,A 88.4814,B 8.3838,C 0.097,E1 8.3917,E2 363.2491} C_DIS
LIN {X 8.2794,Y 135.8932,Z 173,A 86.8048,B 8.3838,C 0.0962,E1 8.3964,E2 364.9183} C_DIS
LIN {X 11.6598,Y 135.645,Z 173,A 85.3642,B 8.3838,C 0.0968,E1 8.4004,E2 366.3601} C_DIS
LIN {X 15.9263,Y 135.2104,Z 173,A 83.7027,B 8.3838,C 0.0948,E1 8.405,E2 368.0037} C_DIS
LIN {X 19.2507,Y 134.7771,Z 173,A 82.1676,B 8.3838,C 0.0975,E1 8.4093,E2 369.5533} C_DIS
LIN {X 23.0908,Y 134.1743,Z 173,A 80.4166,B 8.3838,C 0.1004,E1 8.4141,E2 371.3177} C_DIS
LIN {X 26.9156,Y 133.458,Z 173,A 78.9421,B 8.3838,C 0.0983,E1 8.4181,E2 372.7721} C_DIS
LIN {X 29.5351,Y 132.905,Z 173,A 77.6906,B 8.3838,C 0.1013,E1 8.4216,E2 374.0385} C_DIS
LIN {X 33.2305,Y 132.0274,Z 173,A 76.4191,B 8.3838,C 0.0963,E1 8.4249,E2 375.2699} C_DIS
LIN {X 36.3261,Y 131.2096,Z 173,A 74.9629,B 8.3838,C 0.0993,E1 8.4289,E2 376.739} C_DIS
LIN {X 40.6688,Y 129.9311,Z 173,A 72.8421,B 8.3838,C 0.1049,E1 8.4346,E2 378.8857} C_DIS
LIN {X 44.1752,Y 128.7794,Z 173,A 71.3627,B 8.3838,C 0.1049,E1 8.4385,E2 380.3559} C_DIS
LIN {X 47.1744,Y 127.7119,Z 173,A 69.9699,B 8.3837,C 0.1072,E1 8.4422,E2 381.755} C_DIS
LIN {X 53.0365,Y 125.3909,Z 173,A 67.3151,B 8.3837,C 0.1101,E1 8.449,E2 384.4098} C_DIS
LIN {X 56.9506,Y 123.6609,Z 173,A 65.707,B 8.3837,C 0.1085,E1 8.4531,E2 385.9943} C_DIS
LIN {X 60.1289,Y 122.147,Z 173,A 64.1994,B 8.3837,C 0.1108,E1 8.4569,E2 387.5051} C_DIS
LIN {X 63.1545,Y 120.6104,Z 173,A 62.767,B 8.3837,C 0.1128,E1 8.4604,E2 388.938} C_DIS
LIN {X 66.9949,Y 118.523,Z 173,A 60.8403,B 8.3836,C 0.117,E1 8.4652,E2 390.8754} C_DIS
LIN {X 70.8153,Y 116.281,Z 173,A 58.9889,B 8.3836,C 0.1195,E1 8.4696,E2 392.7254} C_DIS
LIN {X 74.6,Y 113.8896,Z 173,A 57.1213,B 8.3835,C 0.1221,E1 8.474,E2 394.5913} C_DIS
LIN {X 78.2533,Y 111.4109,Z 173,A 55.2725,B 8.3835,C 0.1249,E1 8.4782,E2 396.4391} C_DIS
LIN {X 82.0401,Y 108.6523,Z 173,A 53.4204,B 8.3835,C 0.126,E1 8.4824,E2 398.277} C_DIS
LIN {X 85.3267,Y 106.0909,Z 173,A 51.6108,B 8.3834,C 0.1302,E1 8.4863,E2 400.0938} C_DIS
LIN {X 88.7691,Y 103.2277,Z 173,A 49.8246,B 8.3834,C 0.1317,E1 8.4901,E2 401.8685} C_DIS
LIN {X 91.8961,Y 100.4545,Z 173,A 48.0081,B 8.3833,C 0.1362,E1 8.4939,E2 403.6924} C_DIS
LIN {X 95.1278,Y 97.3996,Z 173,A 46.3,B 8.3833,C 0.1367,E1 8.4973,E2 405.3812} C_DIS
LIN {X 97.4236,Y 95.1033,Z 173,A 44.8326,B 8.3832,C 0.1415,E1 8.5002,E2 406.8613} C_DIS
LIN {X 100.3821,Y 91.9749,Z 173,A 43.0366,B 8.3832,C 0.1449,E1 8.5036,E2 408.6559} C_DIS
LIN {X 103.3957,Y 88.574,Z 173,A 41.1223,B 8.3831,C 0.1491,E1 8.5071,E2 410.5713} C_DIS
LIN {X 105.5844,Y 85.9529,Z 173,A 39.6821,B 8.383,C 0.1524,E1 8.5097,E2 412.0125} C_DIS
LIN {X 108.2233,Y 82.6054,Z 173,A 37.9688,B 8.383,C 0.1548,E1 8.5126,E2 413.7167} C_DIS
LIN {X 110.9187,Y 78.9496,Z 173,A 36.0886,B 8.3829,C 0.1586,E1 8.5157,E2 415.5939} C_DIS
LIN {X 113.445,Y 75.2747,Z 173,A 34.1897,B 8.3828,C 0.1635,E1 8.5187,E2 417.4964} C_DIS
LIN {X 115.8876,Y 71.4568,Z 173,A 32.3182,B 8.3828,C 0.1674,E1 8.5214,E2 419.3645} C_DIS
LIN {X 118.2172,Y 67.5323,Z 173,A 30.4514,B 8.3826,C 0.1711,E1 8.5241,E2 421.2258} C_DIS
LIN {X 120.3293,Y 63.6899,Z 173,A 28.6764,B 8.3826,C 0.1743,E1 8.5264,E2 422.9931} C_DIS
LIN {X 122.1281,Y 60.1672,Z 173,A 27.0967,B 8.3826,C 0.1768,E1 8.5284,E2 424.5633} C_DIS
LIN {X 123.529,Y 57.236,Z 173,A 25.7521,B 8.3825,C 0.1798,E1 8.53,E2 425.906} C_DIS
LIN {X 124.8397,Y 54.3187,Z 173,A 24.4445,B 8.3824,C 0.1826,E1 8.5315,E2 427.2098} C_DIS
LIN {X 126.2227,Y 51.0219,Z 173,A 22.8614,B 8.3823,C 0.1882,E1 8.5331,E2 428.8035} C_DIS
LIN {X 128.4955,Y 44.9942,Z 173,A 20.2472,B 8.3822,C 0.1935,E1 8.5357,E2 431.4076} C_DIS
LIN {X 129.6242,Y 41.6295,Z 173,A 18.879,B 8.3822,C 0.195,E1 8.5369,E2 432.7614} C_DIS
LIN {X 130.7147,Y 38.0673,Z 173,A 17.2291,B 8.382,C 0.201,E1 8.5382,E2 434.4226} C_DIS
LIN {X 131.8525,Y 33.9195,Z 173,A 15.4481,B 8.3819,C 0.2055,E1 8.5395,E2 436.2014} C_DIS
LIN {X 132.6373,Y 30.7071,Z 173,A 14.0497,B 8.3818,C 0.2095,E1 8.5404,E2 437.6017} C_DIS
LIN {X 133.3986,Y 27.2078,Z 173,A 12.6325,B 8.3818,C 0.2119,E1 8.5412,E2 439.009} C_DIS
LIN {X 134.0308,Y 23.8998,Z 173,A 11.2473,B 8.3816,C 0.2152,E1 8.5419,E2 440.3913} C_DIS
LIN {X 134.5417,Y 20.8321,Z 173,A 10.036,B 8.3816,C 0.2169,E1 8.5424,E2 441.5916} C_DIS
LIN {X 135.0763,Y 17.0379,Z 173,A 8.2203,B 8.3814,C 0.2258,E1 8.5431,E2 443.4339} C_DIS
LIN {X 135.5238,Y 12.9918,Z 173,A 6.6633,B 8.3814,C 0.2274,E1 8.5435,E2 444.9729} C_DIS
LIN {X 135.8027,Y 9.6539,Z 173,A 5.2159,B 8.3812,C 0.2323,E1 8.5439,E2 446.4262} C_DIS
LIN {X 136.0174,Y 5.9302,Z 173,A 3.8163,B 8.3812,C 0.2332,E1 8.5441,E2 447.8061} C_DIS
LIN {X 136.117,Y 2.828,Z 173,A 2.5417,B 8.3811,C 0.2363,E1 8.5441,E2 449.078} C_DIS
LIN {X 136.1457,Y -0.5162,Z 173,A 1.0083,B 8.3809,C 0.243,E1 8.5441,E2 450.6284} C_DIS
LIN {X 136.0902,Y -3.8706,Z 173,A -0.2655,B 8.3809,C 0.2442,E1 8.5441,E2 451.8861} C_DIS
LIN {X 135.9248,Y -7.7663,Z 173,A -1.99,B 8.3806,C 0.2507,E1 8.5438,E2 453.6227} C_DIS
LIN {X 135.5957,Y -12.2428,Z 173,A -3.9429,B 8.3804,C 0.2575,E1 8.5434,E2 455.5853} C_DIS
LIN {X 135.1575,Y -16.3705,Z 173,A -5.5268,B 8.3804,C 0.2591,E1 8.5429,E2 457.1505} C_DIS
LIN {X 134.5685,Y -20.659,Z 173,A -7.3232,B 8.3802,C 0.2638,E1 8.5422,E2 458.9454} C_DIS
LIN {X 133.9006,Y -24.6272,Z 173,A -9.0574,B 8.3801,C 0.2695,E1 8.5413,E2 460.6864} C_DIS
LIN {X 133.1355,Y -28.4684,Z 173,A -10.3596,B 8.3801,C 0.2669,E1 8.5406,E2 461.947} C_DIS
LIN {X 132.5656,Y -31.0209,Z 173,A -11.769,B 8.3798,C 0.2766,E1 8.5397,E2 463.3961} C_DIS
LIN {X 131.3025,Y -35.9939,Z 173,A -13.7163,B 8.3798,C 0.2782,E1 8.5384,E2 465.319} C_DIS
LIN {X 130.3134,Y -39.421,Z 173,A -15.2076,B 8.3797,C 0.2822,E1 8.5372,E2 466.8106} C_DIS
LIN {X 129.3791,Y -42.3895,Z 173,A -16.6473,B 8.3794,C 0.2886,E1 8.536,E2 468.2679} C_DIS
LIN {X 128.2722,Y -45.6287,Z 173,A -17.8537,B 8.3794,C 0.2876,E1 8.5349,E2 469.4464} C_DIS
LIN {X 127.0137,Y -49.0205,Z 173,A -19.4736,B 8.3793,C 0.2938,E1 8.5333,E2 471.0801} C_DIS
LIN {X 125.7184,Y -52.2525,Z 173,A -20.8358,B 8.3792,C 0.2956,E1 8.5318,E2 472.4309} C_DIS
LIN {X 124.7088,Y -54.6214,Z 173,A -22.2794,B 8.3788,C 0.3061,E1 8.5302,E2 473.9206} C_DIS
LIN {X 123.274,Y -57.7874,Z 173,A -23.4733,B 8.3788,C 0.3044,E1 8.5288,E2 475.0824} C_DIS
LIN {X 121.837,Y -60.7573,Z 173,A -24.9096,B 8.3788,C 0.309,E1 8.527,E2 476.5261} C_DIS
LIN {X 119.6898,Y -64.8875,Z 173,A -26.8194,B 8.3786,C 0.3131,E1 8.5245,E2 478.4318} C_DIS
LIN {X 117.2148,Y -69.2583,Z 173,A -28.8361,B 8.3784,C 0.3165,E1 8.5217,E2 480.4385} C_DIS
LIN {X 115.0649,Y -72.7736,Z 173,A -30.5315,B 8.3784,C 0.32,E1 8.5192,E2 482.1308} C_DIS
LIN {X 112.6367,Y -76.4782,Z 173,A -32.232,B 8.3783,C 0.3212,E1 8.5166,E2 483.8125} C_DIS
LIN {X 110.5404,Y -79.4786,Z 173,A -33.9461,B 8.378,C 0.3285,E1 8.5138,E2 485.5501} C_DIS
LIN {X 107.8444,Y -83.1001,Z 173,A -35.8815,B 8.3778,C 0.3338,E1 8.5106,E2 487.4918} C_DIS
LIN {X 104.7667,Y -86.9474,Z 173,A -37.8184,B 8.3777,C 0.3357,E1 8.5072,E2 489.4137} C_DIS
LIN {X 101.9644,Y -90.2173,Z 173,A -39.5848,B 8.3776,C 0.3388,E1 8.5039,E2 491.1761} C_DIS
LIN {X 99.1589,Y -93.2923,Z 173,A -41.383,B 8.3774,C 0.3436,E1 8.5005,E2 492.9818} C_DIS
LIN {X 96.2707,Y -96.2707,Z 173,A -43.0721,B 8.3773,C 0.3462,E1 8.4972,E2 494.6655} C_DIS
LIN {X 93.2863,Y -99.1645,Z 173,A -44.8132,B 8.3771,C 0.3497,E1 8.4937,E2 496.4072} C_DIS
LIN {X 90.1906,Y -101.988,Z 173,A -46.5441,B 8.3771,C 0.3525,E1 8.4901,E2 498.1357} C_DIS
LIN {X 86.72,Y -104.955,Z 173,A -48.3987,B 8.3769,C 0.3549,E1 8.4862,E2 499.9837} C_DIS
LIN {X 83.3178,Y -107.6757,Z 173,A -50.2025,B 8.3768,C 0.3578,E1 8.4822,E2 501.7855} C_DIS
LIN {X 80.4248,Y -109.8535,Z 173,A -51.705,B 8.3767,C 0.3601,E1 8.4789,E2 503.2867} C_DIS
LIN {X 77.0002,Y -112.2804,Z 173,A -53.5104,B 8.3765,C 0.364,E1 8.4747,E2 505.0986} C_DIS
LIN {X 73.2716,Y -114.7485,Z 173,A -55.3604,B 8.3765,C 0.3665,E1 8.4704,E2 506.9464} C_DIS
LIN {X 69.4752,Y -117.0862,Z 173,A -56.9933,B 8.3765,C 0.3646,E1 8.4666,E2 508.5501} C_DIS
LIN {X 63.8942,Y -120.222,Z 173,A -59.757,B 8.3763,C 0.3701,E1 8.4598,E2 511.325} C_DIS
LIN {X 60.4265,Y -122.0001,Z 173,A -61.3289,B 8.3763,C 0.3711,E1 8.4559,E2 512.8897} C_DIS
LIN {X 58.0424,Y -123.1542,Z 173,A -62.6771,B 8.3759,C 0.3772,E1 8.4524,E2 514.2683} C_DIS
LIN {X 54.3069,Y -124.8448,Z 173,A -64.2726,B 8.3759,C 0.3768,E1 8.4484,E2 515.8487} C_DIS
LIN {X 51.0434,Y -126.214,Z 173,A -65.7135,B 8.3759,C 0.3777,E1 8.4447,E2 517.2846} C_DIS
LIN {X 48.3051,Y -127.2884,Z 173,A -66.8765,B 8.3759,C 0.3777,E1 8.4417,E2 518.4392} C_DIS
LIN {X 45.6863,Y -128.2514,Z 173,A -68.1271,B 8.3758,C 0.3804,E1 8.4384,E2 519.7003} C_DIS
LIN {X 41.8445,Y -129.5555,Z 173,A -69.8455,B 8.3758,C 0.3824,E1 8.4338,E2 521.4213} C_DIS
LIN {X 38.6954,Y -130.5308,Z 173,A -71.2917,B 8.3756,C 0.3848,E1 8.4299,E2 522.876} C_DIS
LIN {X 35.4749,Y -131.4424,Z 173,A -72.6628,B 8.3756,C 0.3854,E1 8.4262,E2 524.2433} C_DIS
LIN {X 32.1088,Y -132.3046,Z 173,A -74.0747,B 8.3756,C 0.3856,E1 8.4224,E2 525.6499} C_DIS
LIN {X 28.7106,Y -133.0832,Z 173,A -75.4104,B 8.3756,C 0.3842,E1 8.4188,E2 526.9699} C_DIS
LIN {X 26.07,Y -133.6266,Z 173,A -76.537,B 8.3756,C 0.3848,E1 8.4157,E2 528.0962} C_DIS
LIN {X 22.4995,Y -134.273,Z 173,A -78.1583,B 8.3755,C 0.3876,E1 8.4112,E2 529.7304} C_DIS
LIN {X 19.8547,Y -134.6908,Z 173,A -79.2134,B 8.3755,C 0.3868,E1 8.4083,E2 530.7772} C_DIS
LIN {X 16.4594,Y -135.1469,Z 173,A -80.6203,B 8.3755,C 0.3868,E1 8.4045,E2 532.1804} C_DIS
LIN {X 8.5989,Y -135.8735,Z 173,A -85.0635,B 8.3745,C 0.4088,E1 8.3917,E2 536.766} C_DIS
LIN {X 1.3353,Y -136.1399,Z 173,A -87.1249,B 8.3753,C 0.3911,E1 8.3863,E2 538.7042} C_DIS
LIN {X 1.3353,Y -136.1399,Z 173,A -87.1249,B 8.3753,C 0.3911,E1 8.3863,E2 538.7042} C_DIS
Enddeposition()
LIN {X 0.9705,Y -137.0497,Z 173,A -86.8629,B 8.3314,C 0.389,E1 8.3431,E2 538.436} C_DIS
Startdeposition()
$VEL.CP = VEL_PRINT
LIN {X 4.8167,Y -136.97,Z 173,A -85.0144,B 8.3316,C 0.3842,E1 8.3483,E2 536.5559} C_DIS
LIN {X 8.2484,Y -136.8053,Z 173,A -83.6811,B 8.3316,C 0.3857,E1 8.352,E2 535.2351} C_DIS
LIN {X 11.0031,Y -136.6123,Z 173,A -82.5162,B 8.3316,C 0.3852,E1 8.3553,E2 534.0682} C_DIS
LIN {X 13.8792,Y -136.3513,Z 173,A -81.1281,B 8.3318,C 0.3812,E1 8.3592,E2 532.6562} C_DIS
LIN {X 17.271,Y -135.9621,Z 173,A -79.8853,B 8.3317,C 0.3841,E1 8.3626,E2 531.4363} C_DIS
LIN {X 20.1785,Y -135.5623,Z 173,A -78.4851,B 8.3318,C 0.3801,E1 8.3665,E2 530.0131} C_DIS
LIN {X 23.3494,Y -135.0523,Z 173,A -77.2263,B 8.3318,C 0.3809,E1 8.37,E2 528.7644} C_DIS
LIN {X 26.784,Y -134.412,Z 173,A -75.6924,B 8.3319,C 0.3785,E1 8.3742,E2 527.22} C_DIS
LIN {X 30.1929,Y -133.6867,Z 173,A -74.3313,B 8.3319,C 0.3793,E1 8.3779,E2 525.8702} C_DIS
LIN {X 33.1695,Y -132.9802,Z 173,A -73.0417,B 8.3319,C 0.3781,E1 8.3814,E2 524.5784} C_DIS
LIN {X 36.3669,Y -132.1415,Z 173,A -71.7628,B 8.3319,C 0.3789,E1 8.3848,E2 523.3118} C_DIS
LIN {X 39.6133,Y -131.2047,Z 173,A -70.3321,B 8.3319,C 0.3772,E1 8.3886,E2 521.8779} C_DIS
LIN {X 42.7562,Y -130.2146,Z 173,A -68.9864,B 8.3319,C 0.3765,E1 8.3922,E2 520.5352} C_DIS
LIN {X 45.9418,Y -129.1251,Z 173,A -67.4876,B 8.3321,C 0.3732,E1 8.3962,E2 519.0236} C_DIS
LIN {X 49.1172,Y -127.9509,Z 173,A -66.0512,B 8.3322,C 0.3712,E1 8.4,E2 517.5834} C_DIS
LIN {X 52.5117,Y -126.5947,Z 173,A -64.637,B 8.3322,C 0.3716,E1 8.4036,E2 516.1827} C_DIS
LIN {X 55.4244,Y -125.3477,Z 173,A -63.2458,B 8.3323,C 0.3686,E1 8.4072,E2 514.7818} C_DIS
LIN {X 58.5496,Y -123.9188,Z 173,A -61.8193,B 8.3324,C 0.3669,E1 8.4108,E2 513.3555} C_DIS
LIN {X 61.6514,Y -122.4051,Z 173,A -60.3639,B 8.3325,C 0.3646,E1 8.4144,E2 511.8973} C_DIS
LIN {X 64.6055,Y -120.8732,Z 173,A -58.8984,B 8.3327,C 0.3611,E1 8.4181,E2 510.4211} C_DIS
LIN {X 68.2886,Y -118.8317,Z 173,A -57.2263,B 8.3327,C 0.3602,E1 8.4221,E2 508.7589} C_DIS
LIN {X 71.9216,Y -116.6683,Z 173,A -55.4588,B 8.3328,C 0.3574,E1 8.4263,E2 506.9899} C_DIS
LIN {X 75.6153,Y -114.3089,Z 173,A -53.6793,B 8.3329,C 0.3554,E1 8.4305,E2 505.2155} C_DIS
LIN {X 78.7519,Y -112.1711,Z 173,A -52.1237,B 8.333,C 0.3533,E1 8.4341,E2 503.6626} C_DIS
LIN {X 82.094,Y -109.7487,Z 173,A -50.365,B 8.3332,C 0.3495,E1 8.438,E2 501.8979} C_DIS
LIN {X 85.5878,Y -107.0464,Z 173,A -48.5155,B 8.3333,C 0.346,E1 8.4421,E2 500.0464} C_DIS
LIN {X 88.9988,Y -104.2277,Z 173,A -46.7099,B 8.3334,C 0.3433,E1 8.446,E2 498.2448} C_DIS
LIN {X 92.3212,Y -101.2966,Z 173,A -44.8798,B 8.3336,C 0.34,E1 8.4498,E2 496.4157} C_DIS
LIN {X 95.1144,Y -98.6785,Z 173,A -43.3083,B 8.3336,C 0.3373,E1 8.4529,E2 494.8464} C_DIS
LIN {X 98.1594,Y -95.6506,Z 173,A -41.5785,B 8.3338,C 0.3349,E1 8.4563,E2 493.1232} C_DIS
LIN {X 100.6972,Y -92.9746,Z 173,A -40.0569,B 8.3338,C 0.3319,E1 8.4592,E2 491.6027} C_DIS
LIN {X 103.4663,Y -89.8829,Z 173,A -38.2944,B 8.3341,C 0.3275,E1 8.4625,E2 489.835} C_DIS
LIN {X 106.33,Y -86.4763,Z 173,A -36.421,B 8.3342,C 0.3229,E1 8.4658,E2 487.958} C_DIS
LIN {X 109.1334,Y -82.9108,Z 173,A -34.6072,B 8.3343,C 0.3202,E1 8.4689,E2 486.153} C_DIS
LIN {X 111.6628,Y -79.471,Z 173,A -32.8332,B 8.3345,C 0.3161,E1 8.4718,E2 484.3785} C_DIS
LIN {X 113.822,Y -76.3463,Z 173,A -31.3206,B 8.3345,C 0.3138,E1 8.4742,E2 482.874} C_DIS
LIN {X 116.059,Y -72.9007,Z 173,A -29.6144,B 8.3347,C 0.3098,E1 8.4767,E2 481.1675} C_DIS
LIN {X 118.0352,Y -69.6555,Z 173,A -28.0727,B 8.3348,C 0.3068,E1 8.479,E2 479.6301} C_DIS
LIN {X 119.7568,Y -66.6522,Z 173,A -26.5308,B 8.335,C 0.301,E1 8.4811,E2 478.0746} C_DIS
LIN {X 121.7445,Y -62.949,Z 173,A -24.9149,B 8.335,C 0.2995,E1 8.4832,E2 476.475} C_DIS
LIN {X 123.2937,Y -59.858,Z 173,A -23.4936,B 8.3352,C 0.2962,E1 8.4849,E2 475.0553} C_DIS
LIN {X 124.7583,Y -56.7422,Z 173,A -22.0788,B 8.3353,C 0.2929,E1 8.4866,E2 473.6421} C_DIS
LIN {X 126.2425,Y -53.355,Z 173,A -20.5081,B 8.3355,C 0.2882,E1 8.4883,E2 472.0667} C_DIS
LIN {X 127.5602,Y -50.1222,Z 173,A -19.253,B 8.3355,C 0.2886,E1 8.4896,E2 470.8362} C_DIS
LIN {X 128.6428,Y -47.2793,Z 173,A -17.7922,B 8.3357,C 0.281,E1 8.491,E2 469.35} C_DIS
LIN {X 129.7679,Y -44.0975,Z 173,A -16.3502,B 8.3359,C 0.2765,E1 8.4924,E2 467.9026} C_DIS
LIN {X 130.9135,Y -40.5649,Z 173,A -14.9941,B 8.3359,C 0.2764,E1 8.4935,E2 466.57} C_DIS
LIN {X 131.7654,Y -37.712,Z 173,A -13.7435,B 8.336,C 0.2728,E1 8.4945,E2 465.3175} C_DIS
LIN {X 132.6388,Y -34.5146,Z 173,A -12.3836,B 8.3361,C 0.2694,E1 8.4954,E2 463.9595} C_DIS
LIN {X 133.4876,Y -31.0647,Z 173,A -11.0203,B 8.3361,C 0.2678,E1 8.4963,E2 462.6102} C_DIS
LIN {X 134.2463,Y -27.5981,Z 173,A -9.5522,B 8.3363,C 0.2639,E1 8.4972,E2 461.1425} C_DIS
LIN {X 134.8129,Y -24.687,Z 173,A -8.3462,B 8.3363,C 0.2611,E1 8.4978,E2 459.9398} C_DIS
LIN {X 135.356,Y -21.5112,Z 173,A -6.9319,B 8.3365,C 0.2558,E1 8.4984,E2 458.5156} C_DIS
LIN {X 135.7882,Y -18.5978,Z 173,A -5.5893,B 8.3367,C 0.2499,E1 8.499,E2 457.1577} C_DIS
LIN {X 136.2093,Y -15.1991,Z 173,A -4.3196,B 8.3367,C 0.2492,E1 8.4994,E2 455.9071} C_DIS
LIN {X 136.5015,Y -12.3151,Z 173,A -3.1301,B 8.3368,C 0.2462,E1 8.4997,E2 454.7194} C_DIS
LIN {X 136.7507,Y -9.1353,Z 173,A -1.8467,B 8.3369,C 0.2434,E1 8.5,E2 453.4411} C_DIS
LIN {X 136.9196,Y -6.11,Z 173,A -0.5042,B 8.3371,C 0.2381,E1 8.5001,E2 452.0878} C_DIS
LIN {X 137.0475,Y -1.5177,Z 173,A 1.3592,B 8.3371,C 0.2338,E1 8.5002,E2 450.23} C_DIS
LIN {X 137.0221,Y 3.0421,Z 173,A 3.2556,B 8.3373,C 0.2285,E1 8.5002,E2 448.3331} C_DIS
LIN {X 136.9073,Y 6.3547,Z 173,A 4.5433,B 8.3373,C 0.2266,E1 8.5,E2 447.0565} C_DIS
LIN {X 136.7286,Y 9.4482,Z 173,A 5.9059,B 8.3375,C 0.2214,E1 8.4998,E2 445.6843} C_DIS
LIN {X 136.5015,Y 12.3151,Z 173,A 7.0024,B 8.3375,C 0.2202,E1 8.4995,E2 444.6002} C_DIS
LIN {X 136.1825,Y 15.4479,Z 173,A 8.3777,B 8.3377,C 0.2152,E1 8.4991,E2 443.2163} C_DIS
LIN {X 135.7882,Y 18.5978,Z 173,A 9.6049,B 8.3377,C 0.2135,E1 8.4987,E2 442.0006} C_DIS
LIN {X 135.2751,Y 22.0141,Z 173,A 11.069,B 8.3378,C 0.209,E1 8.498,E2 440.5328} C_DIS
LIN {X 134.6574,Y 25.5163,Z 173,A 12.4662,B 8.3378,C 0.2067,E1 8.4973,E2 439.1457} C_DIS
LIN {X 134.0844,Y 28.3783,Z 173,A 13.5973,B 8.3379,C 0.2051,E1 8.4967,E2 438.0249} C_DIS
LIN {X 133.3686,Y 31.5714,Z 173,A 15.0927,B 8.3381,C 0.1986,E1 8.4957,E2 436.5123} C_DIS
LIN {X 132.4788,Y 35.1144,Z 173,A 16.5523,B 8.3381,C 0.1957,E1 8.4947,E2 435.0601} C_DIS
LIN {X 131.6537,Y 38.0933,Z 173,A 17.6701,B 8.3381,C 0.1959,E1 8.4939,E2 433.9633} C_DIS
LIN {X 130.8086,Y 40.9074,Z 173,A 19.109,B 8.3383,C 0.188,E1 8.4927,E2 432.4971} C_DIS
LIN {X 129.6484,Y 44.4422,Z 173,A 20.5271,B 8.3383,C 0.1867,E1 8.4915,E2 431.0951} C_DIS
LIN {X 128.5486,Y 47.531,Z 173,A 21.9071,B 8.3385,C 0.1828,E1 8.4901,E2 429.7131} C_DIS
LIN {X 127.3395,Y 50.6813,Z 173,A 23.205,B 8.3385,C 0.1814,E1 8.4888,E2 428.4284} C_DIS
LIN {X 126.0304,Y 53.8541,Z 173,A 24.7099,B 8.3385,C 0.1761,E1 8.4872,E2 426.9137} C_DIS
LIN {X 124.6046,Y 57.0745,Z 173,A 26.1888,B 8.3387,C 0.1721,E1 8.4855,E2 425.433} C_DIS
LIN {X 123.1725,Y 60.1036,Z 173,A 27.5407,B 8.3387,C 0.1695,E1 8.4839,E2 424.0864} C_DIS
LIN {X 121.6167,Y 63.1925,Z 173,A 29.0258,B 8.3388,C 0.165,E1 8.482,E2 422.5955} C_DIS
LIN {X 119.6224,Y 66.8932,Z 173,A 30.8066,B 8.3389,C 0.1601,E1 8.4796,E2 420.8109} C_DIS
LIN {X 117.4338,Y 70.6648,Z 173,A 32.6115,B 8.3389,C 0.156,E1 8.477,E2 419.0073} C_DIS
LIN {X 114.9692,Y 74.607,Z 173,A 34.4811,B 8.339,C 0.1528,E1 8.4742,E2 417.146} C_DIS
LIN {X 112.6745,Y 78.0299,Z 173,A 36.1103,B 8.339,C 0.1507,E1 8.4717,E2 415.5276} C_DIS
LIN {X 110.2749,Y 81.3858,Z 173,A 37.8631,B 8.3392,C 0.1461,E1 8.4688,E2 413.7705} C_DIS
LIN {X 107.5963,Y 84.8955,Z 173,A 39.6843,B 8.3392,C 0.1424,E1 8.4657,E2 411.9516} C_DIS
LIN {X 104.8005,Y 88.3236,Z 173,A 41.5438,B 8.3393,C 0.1381,E1 8.4623,E2 410.0901} C_DIS
LIN {X 101.8658,Y 91.6929,Z 173,A 43.3129,B 8.3393,C 0.1361,E1 8.4591,E2 408.3326} C_DIS
LIN {X 99.292,Y 94.4738,Z 173,A 44.8665,B 8.3393,C 0.1335,E1 8.4561,E2 406.7823} C_DIS
LIN {X 96.3837,Y 97.4392,Z 173,A 46.5972,B 8.3394,C 0.13,E1 8.4527,E2 405.0518} C_DIS
LIN {X 93.6241,Y 100.0936,Z 173,A 48.1631,B 8.3394,C 0.1276,E1 8.4496,E2 403.4897} C_DIS
LIN {X 90.5499,Y 102.883,Z 173,A 49.9532,B 8.3395,C 0.1232,E1 8.4458,E2 401.6924} C_DIS
LIN {X 87.1793,Y 105.7543,Z 173,A 51.7597,B 8.3395,C 0.1207,E1 8.442,E2 399.891} C_DIS
LIN {X 83.7231,Y 108.5111,Z 173,A 53.6175,B 8.3396,C 0.1172,E1 8.4379,E2 398.0316} C_DIS
LIN {X 80.1872,Y 111.1495,Z 173,A 55.3763,B 8.3396,C 0.1158,E1 8.4339,E2 396.2832} C_DIS
LIN {X 77.0747,Y 113.33,Z 173,A 57.0167,B 8.3396,C 0.1122,E1 8.4301,E2 394.6362} C_DIS
LIN {X 73.5007,Y 115.6803,Z 173,A 58.8268,B 8.3397,C 0.109,E1 8.4259,E2 392.8232} C_DIS
LIN {X 69.7958,Y 117.9527,Z 173,A 60.5382,B 8.3397,C 0.1084,E1 8.4218,E2 391.1248} C_DIS
LIN {X 66.2112,Y 120.001,Z 173,A 62.2957,B 8.3397,C 0.1054,E1 8.4175,E2 389.3632} C_DIS
LIN {X 62.949,Y 121.7445,Z 173,A 63.7453,B 8.3397,C 0.1052,E1 8.414,E2 387.9257} C_DIS
LIN {X 59.858,Y 123.2937,Z 173,A 65.3244,B 8.3398,C 0.1008,E1 8.41,E2 386.33} C_DIS
LIN {X 56.3367,Y 124.9397,Z 173,A 66.8171,B 8.3398,C 0.1014,E1 8.4062,E2 384.8538} C_DIS
LIN {X 53.355,Y 126.2425,Z 173,A 68.1392,B 8.3398,C 0.1006,E1 8.4029,E2 383.5364} C_DIS
LIN {X 50.4495,Y 127.4329,Z 173,A 69.4425,B 8.3398,C 0.0994,E1 8.3995,E2 382.2345} C_DIS
LIN {X 47.2793,Y 128.6428,Z 173,A 70.9357,B 8.3398,C 0.0966,E1 8.3955,E2 380.7322} C_DIS
LIN {X 43.6577,Y 129.9144,Z 173,A 72.3842,B 8.3398,C 0.098,E1 8.3918,E2 379.3031} C_DIS
LIN {X 40.4764,Y 130.9405,Z 173,A 73.7759,B 8.3398,C 0.0969,E1 8.3881,E2 377.9124} C_DIS
LIN {X 37.712,Y 131.7654,Z 173,A 75.0311,B 8.3399,C 0.0951,E1 8.3847,E2 376.6514} C_DIS
LIN {X 34.0665,Y 132.7525,Z 173,A 76.6177,B 8.3399,C 0.0938,E1 8.3804,E2 375.0641} C_DIS
LIN {X 31.0647,Y 133.4876,Z 173,A 77.7892,B 8.3399,C 0.0952,E1 8.3773,E2 373.9078} C_DIS
LIN {X 28.1252,Y 134.139,Z 173,A 79.22,B 8.3399,C 0.0912,E1 8.3733,E2 372.4561} C_DIS
LIN {X 24.4627,Y 134.853,Z 173,A 80.718,B 8.3399,C 0.0916,E1 8.3692,E2 370.9661} C_DIS
LIN {X 21.1516,Y 135.4116,Z 173,A 81.9802,B 8.3399,C 0.0935,E1 8.3658,E2 369.7218} C_DIS
LIN {X 18.5978,Y 135.7882,Z 173,A 83.3219,B 8.3399,C 0.0883,E1 8.362,E2 368.3482} C_DIS
LIN {X 15.1991,Y 136.2093,Z 173,A 84.5884,B 8.3399,C 0.0909,E1 8.3585,E2 367.1025} C_DIS
LIN {X 12.3151,Y 136.5015,Z 173,A 85.7969,B 8.3399,C 0.0906,E1 8.3552,E2 365.8949} C_DIS
LIN {X 8.8038,Y 136.7711,Z 173,A 87.1165,B 8.3399,C 0.0931,E1 8.3515,E2 364.5945} C_DIS
LIN {X 5.7035,Y 136.9354,Z 173,A 88.5086,B 8.3399,C 0.0912,E1 8.3476,E2 363.1915} C_DIS
LIN {X 3.0421,Y 137.0221,Z 173,A 89.7464,B 8.3399,C 0.0889,E1 8.3441,E2 361.9389} C_DIS
LIN {X 0,Y 137.0559,Z 173,A 91.0177,B 8.3399,C 0.0889,E1 8.3406,E2 360.6682} C_DIS
LIN {X -3.0421,Y 137.0221,Z 173,A 92.2933,B 8.3399,C 0.0889,E1 8.337,E2 359.3927} C_DIS
LIN {X -6.3547,Y 136.9073,Z 173,A 93.6045,B 8.3399,C 0.0904,E1 8.3334,E2 358.0913} C_DIS
LIN {X -9.4482,Y 136.7286,Z 173,A 94.9042,B 8.3399,C 0.0906,E1 8.3298,E2 356.7917} C_DIS
LIN {X -12.3151,Y 136.5015,Z 173,A 96.1104,B 8.3399,C 0.0909,E1 8.3264,E2 355.5858} C_DIS
LIN {X -15.4479,Y 136.1825,Z 173,A 97.513,B 8.3399,C 0.0898,E1 8.3225,E2 354.1733} C_DIS
LIN {X -19.182,Y 135.7047,Z 173,A 99.0121,B 8.3399,C 0.0917,E1 8.3184,E2 352.6842} C_DIS
LIN {X -22.0141,Y 135.2751,Z 173,A 100.1195,B 8.3399,C 0.0938,E1 8.3153,E2 351.5886} C_DIS
LIN {X -24.9391,Y 134.7678,Z 173,A 101.5455,B 8.3399,C 0.0913,E1 8.3114,E2 350.1407} C_DIS
LIN {X -28.3783,Y 134.0844,Z 173,A 102.8388,B 8.3399,C 0.0951,E1 8.3079,E2 348.8694} C_DIS
LIN {X -31.6122,Y 133.3588,Z 173,A 104.3915,B 8.3399,C 0.0932,E1 8.3036,E2 347.297} C_DIS
LIN {X -34.7681,Y 132.5712,Z 173,A 105.6972,B 8.3399,C 0.0951,E1 8.3001,E2 345.9989} C_DIS
LIN {X -37.712,Y 131.7654,Z 173,A 107.1324,B 8.3399,C 0.0934,E1 8.2962,E2 344.5451} C_DIS
LIN {X -41.4434,Y 130.6374,Z 173,A 108.6273,B 8.3399,C 0.0971,E1 8.2922,E2 343.0677} C_DIS
LIN {X -44.0975,Y 129.7679,Z 173,A 109.8843,B 8.3399,C 0.0967,E1 8.2889,E2 341.8006} C_DIS
LIN {X -47.531,Y 128.5486,Z 173,A 111.3325,B 8.3399,C 0.0995,E1 8.2851,E2 340.3627} C_DIS
LIN {X -50.4495,Y 127.4329,Z 173,A 112.6486,B 8.3399,C 0.1007,E1 8.2817,E2 339.0465} C_DIS
LIN {X -53.8541,Y 126.0304,Z 173,A 114.2273,B 8.3399,C 0.1018,E1 8.2776,E2 337.4641} C_DIS
LIN {X -56.9897,Y 124.6438,Z 173,A 115.6459,B 8.3398,C 0.1038,E1 8.274,E2 336.0485} C_DIS
LIN {X -60.1036,Y 123.1725,Z 173,A 117.0984,B 8.3398,C 0.1054,E1 8.2704,E2 334.5955} C_DIS
LIN {X -63.1925,Y 121.6167,Z 173,A 118.6302,B 8.3398,C 0.1059,E1 8.2665,E2 333.0542} C_DIS
LIN {X -66.8932,Y 119.6224,Z 173,A 120.4435,B 8.3398,C 0.1074,E1 8.2621,E2 331.2356} C_DIS
LIN {X -70.6648,Y 117.4338,Z 173,A 122.1726,B 8.3397,C 0.1117,E1 8.258,E2 329.5196} C_DIS
LIN {X -73.6412,Y 115.5906,Z 173,A 123.7641,B 8.3397,C 0.1119,E1 8.2542,E2 327.9136} C_DIS
LIN {X -77.2735,Y 113.1947,Z 173,A 125.4996,B 8.3397,C 0.1162,E1 8.2502,E2 326.19} C_DIS
LIN {X -80.1872,Y 111.1495,Z 173,A 127.1078,B 8.3397,C 0.1168,E1 8.2465,E2 324.5683} C_DIS
LIN {X -83.7231,Y 108.5111,Z 173,A 128.9735,B 8.3396,C 0.1197,E1 8.2423,E2 322.7017} C_DIS
LIN {X -87.1793,Y 105.7543,Z 173,A 130.8436,B 8.3396,C 0.1228,E1 8.2383,E2 320.8305} C_DIS
LIN {X -90.5499,Y 102.883,Z 173,A 132.7172,B 8.3395,C 0.126,E1 8.2343,E2 318.9558} C_DIS
LIN {X -93.8294,Y 99.9012,Z 173,A 134.4791,B 8.3395,C 0.1311,E1 8.2307,E2 317.2069} C_DIS
LIN {X -96.3837,Y 97.4392,Z 173,A 136.0962,B 8.3395,C 0.132,E1 8.2275,E2 315.5747} C_DIS
LIN {X -99.3892,Y 94.3722,Z 173,A 137.8366,B 8.3393,C 0.1366,E1 8.2241,E2 313.8429} C_DIS
LIN {X -101.8916,Y 91.6641,Z 173,A 139.4758,B 8.3393,C 0.1384,E1 8.221,E2 312.193} C_DIS
LIN {X -104.8005,Y 88.3236,Z 173,A 141.3528,B 8.3393,C 0.1421,E1 8.2176,E2 310.3148} C_DIS
LIN {X -107.5963,Y 84.8955,Z 173,A 143.2275,B 8.3392,C 0.1459,E1 8.2143,E2 308.4387} C_DIS
LIN {X -110.2749,Y 81.3858,Z 173,A 145.099,B 8.3392,C 0.1498,E1 8.2112,E2 306.5658} C_DIS
LIN {X -112.8331,Y 77.8003,Z 173,A 146.8532,B 8.339,C 0.1556,E1 8.2084,E2 304.8243} C_DIS
LIN {X -115.0046,Y 74.5524,Z 173,A 148.5592,B 8.339,C 0.1584,E1 8.2058,E2 303.1109} C_DIS
LIN {X -117.0532,Y 71.2942,Z 173,A 150.1432,B 8.3389,C 0.1628,E1 8.2034,E2 301.5316} C_DIS
LIN {X -119.0934,Y 67.8299,Z 173,A 151.9332,B 8.3389,C 0.1654,E1 8.2009,E2 299.7298} C_DIS
LIN {X -120.9384,Y 64.4842,Z 173,A 153.4706,B 8.3387,C 0.1704,E1 8.1989,E2 298.2014} C_DIS
LIN {X -122.5296,Y 61.4068,Z 173,A 154.9411,B 8.3387,C 0.1738,E1 8.197,E2 296.7296} C_DIS
LIN {X -124.0366,Y 58.303,Z 173,A 156.4058,B 8.3386,C 0.1773,E1 8.1953,E2 295.2636} C_DIS
LIN {X -125.4588,Y 55.176,Z 173,A 157.9526,B 8.3386,C 0.1794,E1 8.1935,E2 293.7045} C_DIS
LIN {X -126.9942,Y 51.5378,Z 173,A 159.3404,B 8.3383,C 0.1878,E1 8.192,E2 292.3508} C_DIS
LIN {X -128.0485,Y 48.8661,Z 173,A 160.7604,B 8.3383,C 0.1878,E1 8.1906,E2 290.905} C_DIS
LIN {X -129.3035,Y 45.4372,Z 173,A 162.2103,B 8.3383,C 0.1931,E1 8.1892,E2 289.4662} C_DIS
LIN {X -130.3796,Y 42.2502,Z 173,A 163.8002,B 8.3382,C 0.1942,E1 8.1878,E2 287.8548} C_DIS
LIN {X -131.3717,Y 39.0567,Z 173,A 165.0603,B 8.3381,C 0.2001,E1 8.1868,E2 286.6132} C_DIS
LIN {X -132.2125,Y 36.1134,Z 173,A 166.4607,B 8.3381,C 0.2019,E1 8.1857,E2 285.1992} C_DIS
LIN {X -133.0445,Y 32.916,Z 173,A 167.9489,B 8.338,C 0.2042,E1 8.1847,E2 283.699} C_DIS
LIN {X -133.9098,Y 29.1869,Z 173,A 169.2835,B 8.3377,C 0.2127,E1 8.1839,E2 282.3989} C_DIS
LIN {X -134.5117,Y 26.2787,Z 173,A 170.7514,B 8.3377,C 0.2129,E1 8.1831,E2 280.9041} C_DIS
LIN {X -135.0523,Y 23.3494,Z 173,A 172.1004,B 8.3377,C 0.2149,E1 8.1824,E2 279.5435} C_DIS
LIN {X -135.5981,Y 19.9278,Z 173,A 173.5738,B 8.3376,C 0.2186,E1 8.1818,E2 278.0684} C_DIS
LIN {X -136.0524,Y 16.5381,Z 173,A 174.8693,B 8.3374,C 0.2248,E1 8.1813,E2 276.7909} C_DIS
LIN {X -136.3751,Y 13.6311,Z 173,A 176.0902,B 8.3374,C 0.2283,E1 8.181,E2 275.5715} C_DIS
LIN {X -136.6339,Y 10.7453,Z 173,A 177.4113,B 8.3373,C 0.2302,E1 8.1807,E2 274.2378} C_DIS
LIN {X -136.842,Y 7.653,Z 173,A 178.8875,B 8.3373,C 0.2312,E1 8.1804,E2 272.7402} C_DIS
LIN {X -136.9996,Y 3.8503,Z 173,A -179.609,B 8.3371,C 0.2371,E1 8.1803,E2 271.2491} C_DIS
LIN {X -137.0572,Y 0,Z 173,A -177.8944,B 8.3371,C 0.2402,E1 8.1803,E2 269.5229} C_DIS
LIN {X -137.0221,Y -3.0421,Z 173,A -176.6369,B 8.3369,C 0.2441,E1 8.1803,E2 268.2683} C_DIS
LIN {X -136.9073,Y -6.3547,Z 173,A -175.2285,B 8.3368,C 0.2477,E1 8.1805,E2 266.8583} C_DIS
LIN {X -136.6946,Y -9.9148,Z 173,A -173.7576,B 8.3366,C 0.2523,E1 8.1808,E2 265.3911} C_DIS
LIN {X -136.3513,Y -13.8792,Z 173,A -172.086,B 8.3366,C 0.257,E1 8.1812,E2 263.7201} C_DIS
LIN {X -135.9621,Y -17.271,Z 173,A -170.5817,B 8.3364,C 0.2599,E1 8.1817,E2 262.2073} C_DIS
LIN {X -135.4845,Y -20.681,Z 173,A -169.155,B 8.3363,C 0.2642,E1 8.1823,E2 260.7833} C_DIS
LIN {X -134.7678,Y -24.9391,Z 173,A -167.1939,B 8.3362,C 0.267,E1 8.1832,E2 258.8041} C_DIS
LIN {X -134.0579,Y -28.5011,Z 173,A -165.714,B 8.336,C 0.2718,E1 8.1841,E2 257.3302} C_DIS
LIN {X -133.2977,Y -31.8657,Z 173,A -164.3981,B 8.3358,C 0.2778,E1 8.1849,E2 256.0312} C_DIS
LIN {X -132.5712,Y -34.7681,Z 173,A -163.0313,B 8.3358,C 0.2795,E1 8.1858,E2 254.6509} C_DIS
LIN {X -131.7654,Y -37.712,Z 173,A -161.7315,B 8.3357,C 0.2826,E1 8.1868,E2 253.3491} C_DIS
LIN {X -130.8086,Y -40.9074,Z 173,A -160.1953,B 8.3357,C 0.2843,E1 8.1881,E2 251.7961} C_DIS
LIN {X -129.7679,Y -44.0975,Z 173,A -158.7954,B 8.3355,C 0.2881,E1 8.1894,E2 250.3975} C_DIS
LIN {X -128.5486,Y -47.531,Z 173,A -157.2909,B 8.3353,C 0.2925,E1 8.1908,E2 248.8964} C_DIS
LIN {X -127.4329,Y -50.4495,Z 173,A -155.8535,B 8.3353,C 0.294,E1 8.1923,E2 247.4433} C_DIS
LIN {X -125.9901,Y -53.9472,Z 173,A -154.3677,B 8.3351,C 0.2996,E1 8.1939,E2 245.9706} C_DIS
LIN {X -124.6438,Y -56.9897,Z 173,A -152.9784,B 8.335,C 0.3033,E1 8.1955,E2 244.5824} C_DIS
LIN {X -123.1014,Y -60.2477,Z 173,A -151.413,B 8.3349,C 0.3062,E1 8.1974,E2 243.0105} C_DIS
LIN {X -121.6167,Y -63.1925,Z 173,A -150.1058,B 8.3347,C 0.3108,E1 8.199,E2 241.7133} C_DIS
LIN {X -119.7193,Y -66.72,Z 173,A -148.336,B 8.3346,C 0.3135,E1 8.2014,E2 239.9324} C_DIS
LIN {X -117.8818,Y -69.9148,Z 173,A -146.6643,B 8.3346,C 0.3152,E1 8.2038,E2 238.245} C_DIS
LIN {X -115.5906,Y -73.6412,Z 173,A -144.8066,B 8.3344,C 0.3192,E1 8.2065,E2 236.3845} C_DIS
LIN {X -113.2096,Y -77.2518,Z 173,A -142.9612,B 8.3342,C 0.3228,E1 8.2094,E2 234.5353} C_DIS
LIN {X -110.5668,Y -80.9884,Z 173,A -141.054,B 8.3341,C 0.3273,E1 8.2125,E2 232.6297} C_DIS
LIN {X -108.0556,Y -84.3107,Z 173,A -139.3399,B 8.3339,C 0.3316,E1 8.2154,E2 230.9198} C_DIS
LIN {X -105.3408,Y -87.6787,Z 173,A -137.4806,B 8.3338,C 0.3347,E1 8.2187,E2 229.0548} C_DIS
Enddeposition()
END
